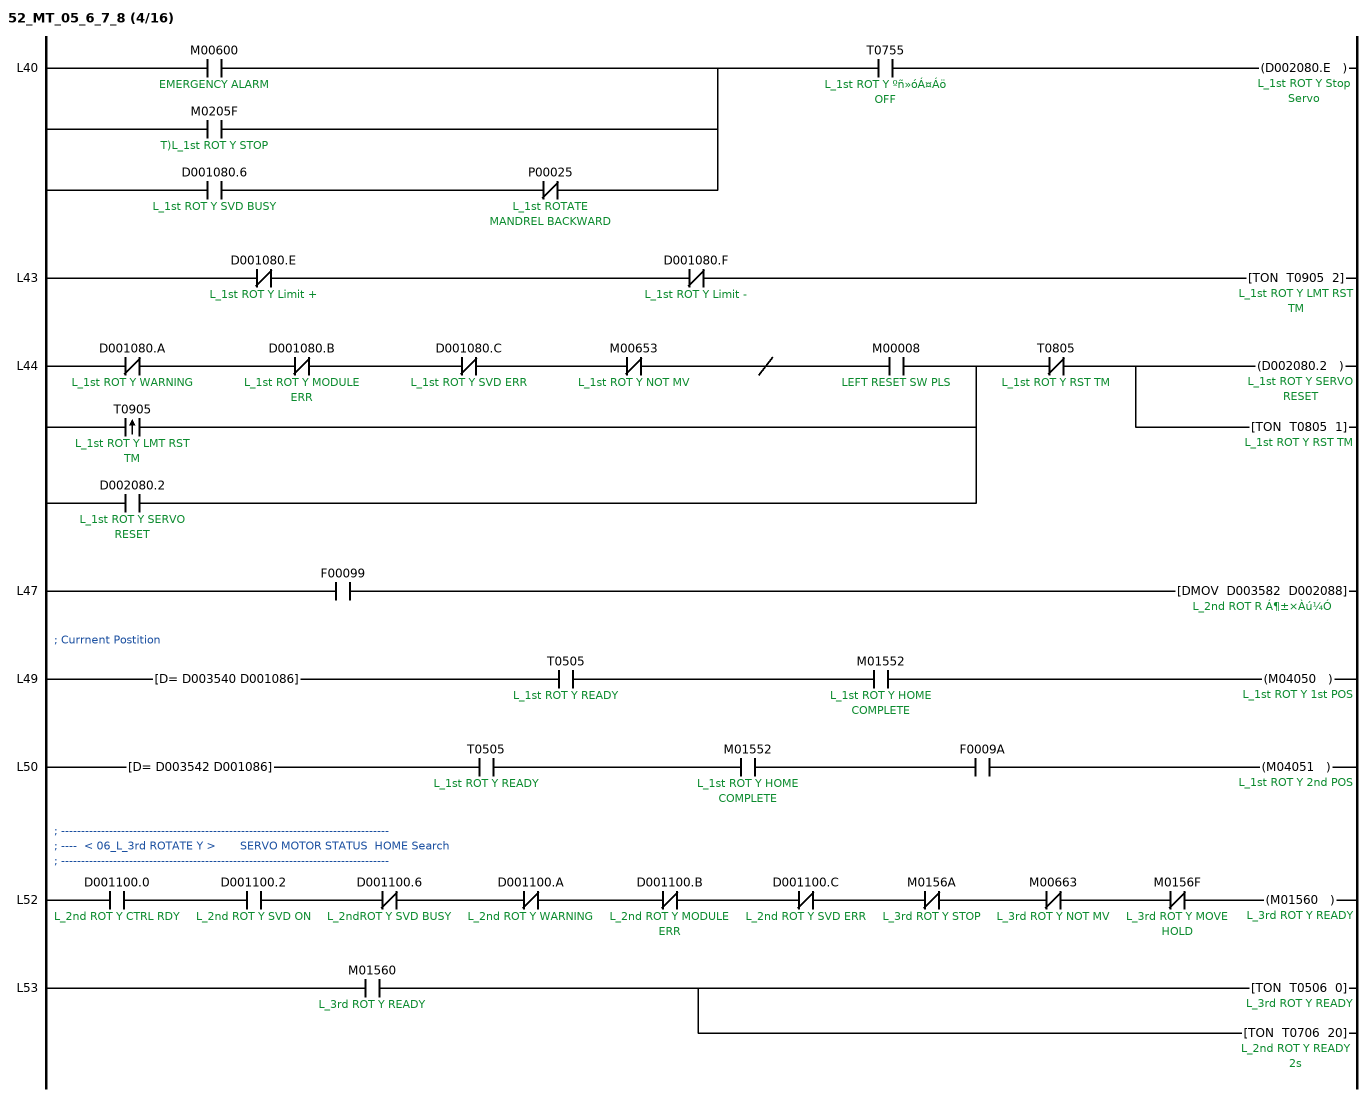
[picture p264: 52_MT_05_6_7_8 rungs L40-L53]
; L40
LOAD      M00600	// EMERGENCY ALARM
OR        M0205F	// T)L_1st ROT Y STOP
LOAD      D001080.6	// L_1st ROT Y SVD BUSY
AND NOT   P00025	// L_1st ROTATE MANDREL BACKWARD
OR LOAD
AND       T0755	// L_1st ROT Y ºñ»óÁ¤Áö OFF
OUT       D002080.E	// L_1st ROT Y Stop Servo
; L43
LOAD NOT  D001080.E	// L_1st ROT Y Limit +
AND NOT   D001080.F	// L_1st ROT Y Limit -
TON       T0905 2	// L_1st ROT Y LMT RST TM
; L44
LOAD NOT  D001080.A	// L_1st ROT Y WARNING
AND NOT   D001080.B	// L_1st ROT Y MODULE ERR
AND NOT   D001080.C	// L_1st ROT Y SVD ERR
AND NOT   M00653	// L_1st ROT Y NOT MV
NOT
AND       M00008	// LEFT RESET SW PLS
ORP       T0905	// L_1st ROT Y LMT RST TM
OR        D002080.2	// L_1st ROT Y SERVO RESET
AND NOT   T0805	// L_1st ROT Y RST TM
OUT       D002080.2	// L_1st ROT Y SERVO RESET
TON       T0805 1	// L_1st ROT Y RST TM
; L47
LOAD      F00099
DMOV      D003582 D002088	// L_2nd ROT R Á¶±×Àú¼Ó
// Currnent Postition
; L49
LOADD=    D003540 D001086
AND       T0505	// L_1st ROT Y READY
AND       M01552	// L_1st ROT Y HOME COMPLETE
OUT       M04050	// L_1st ROT Y 1st POS
; L50
LOADD=    D003542 D001086
AND       T0505	// L_1st ROT Y READY
AND       M01552	// L_1st ROT Y HOME COMPLETE
AND       F0009A
OUT       M04051	// L_1st ROT Y 2nd POS
// ----------------------------------------------------------------------------------
// 
// ----  < 06_L_3rd ROTATE Y >       SERVO MOTOR STATUS  HOME Search
// 
// ----------------------------------------------------------------------------------
; L52
LOAD      D001100.0	// L_2nd ROT Y CTRL RDY
AND       D001100.2	// L_2nd ROT Y SVD ON
AND NOT   D001100.6	// L_2ndROT Y SVD BUSY
AND NOT   D001100.A	// L_2nd ROT Y WARNING
AND NOT   D001100.B	// L_2nd ROT Y MODULE ERR
AND NOT   D001100.C	// L_2nd ROT Y SVD ERR
AND NOT   M0156A	// L_3rd ROT Y STOP
AND NOT   M00663	// L_3rd ROT Y NOT MV
AND NOT   M0156F	// L_3rd ROT Y MOVE HOLD
OUT       M01560	// L_3rd ROT Y READY
; L53
LOAD      M01560	// L_3rd ROT Y READY
TON       T0506 0	// L_3rd ROT Y READY
TON       T0706 20	// L_2nd ROT Y READY 2s

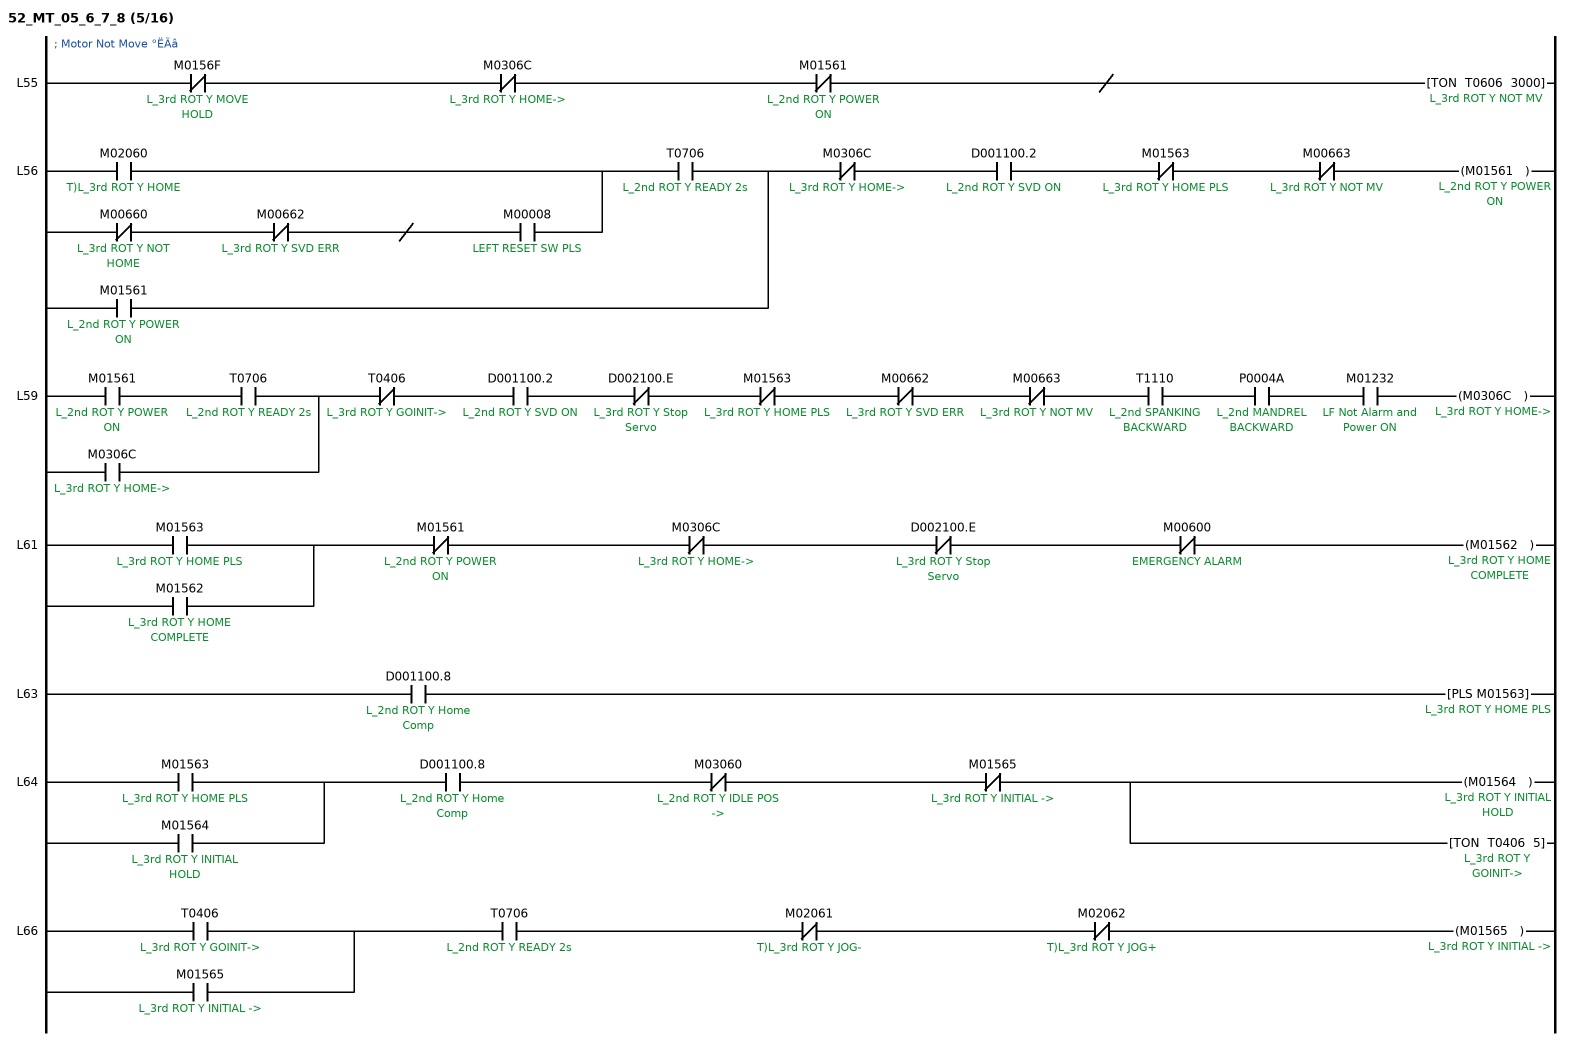
; L55
LOAD NOT  M0156F	// L_3rd ROT Y MOVE HOLD
AND NOT   M0306C	// L_3rd ROT Y HOME->
AND NOT   M01561	// L_2nd ROT Y POWER ON
NOT
TON       T0606 3000	// L_3rd ROT Y NOT MV
// output comment: Motor Not Move °ËÃâ
; L56
LOAD      M02060	// T)L_3rd ROT Y HOME
LOAD NOT  M00660	// L_3rd ROT Y NOT HOME
AND NOT   M00662	// L_3rd ROT Y SVD ERR
NOT
AND       M00008	// LEFT RESET SW PLS
OR LOAD
AND       T0706	// L_2nd ROT Y READY 2s
OR        M01561	// L_2nd ROT Y POWER ON
AND NOT   M0306C	// L_3rd ROT Y HOME->
AND       D001100.2	// L_2nd ROT Y SVD ON
AND NOT   M01563	// L_3rd ROT Y HOME PLS
AND NOT   M00663	// L_3rd ROT Y NOT MV
OUT       M01561	// L_2nd ROT Y POWER ON
; L59
LOAD      M01561	// L_2nd ROT Y POWER ON
AND       T0706	// L_2nd ROT Y READY 2s
OR        M0306C	// L_3rd ROT Y HOME->
AND NOT   T0406	// L_3rd ROT Y GOINIT->
AND       D001100.2	// L_2nd ROT Y SVD ON
AND NOT   D002100.E	// L_3rd ROT Y Stop Servo
AND NOT   M01563	// L_3rd ROT Y HOME PLS
AND NOT   M00662	// L_3rd ROT Y SVD ERR
AND NOT   M00663	// L_3rd ROT Y NOT MV
AND       T1110	// L_2nd SPANKING BACKWARD
AND       P0004A	// L_2nd MANDREL BACKWARD
AND       M01232	// LF Not Alarm and Power ON
OUT       M0306C	// L_3rd ROT Y HOME->
; L61
LOAD      M01563	// L_3rd ROT Y HOME PLS
OR        M01562	// L_3rd ROT Y HOME COMPLETE
AND NOT   M01561	// L_2nd ROT Y POWER ON
AND NOT   M0306C	// L_3rd ROT Y HOME->
AND NOT   D002100.E	// L_3rd ROT Y Stop Servo
AND NOT   M00600	// EMERGENCY ALARM
OUT       M01562	// L_3rd ROT Y HOME COMPLETE
; L63
LOAD      D001100.8	// L_2nd ROT Y Home Comp
OUTP      M01563	// L_3rd ROT Y HOME PLS
; L64
LOAD      M01563	// L_3rd ROT Y HOME PLS
OR        M01564	// L_3rd ROT Y INITIAL HOLD
AND       D001100.8	// L_2nd ROT Y Home Comp
AND NOT   M03060	// L_2nd ROT Y IDLE POS ->
AND NOT   M01565	// L_3rd ROT Y INITIAL ->
OUT       M01564	// L_3rd ROT Y INITIAL HOLD
TON       T0406 5	// L_3rd ROT Y GOINIT->
; L66
LOAD      T0406	// L_3rd ROT Y GOINIT->
OR        M01565	// L_3rd ROT Y INITIAL ->
AND       T0706	// L_2nd ROT Y READY 2s
AND NOT   M02061	// T)L_3rd ROT Y JOG-
AND NOT   M02062	// T)L_3rd ROT Y JOG+
OUT       M01565	// L_3rd ROT Y INITIAL ->

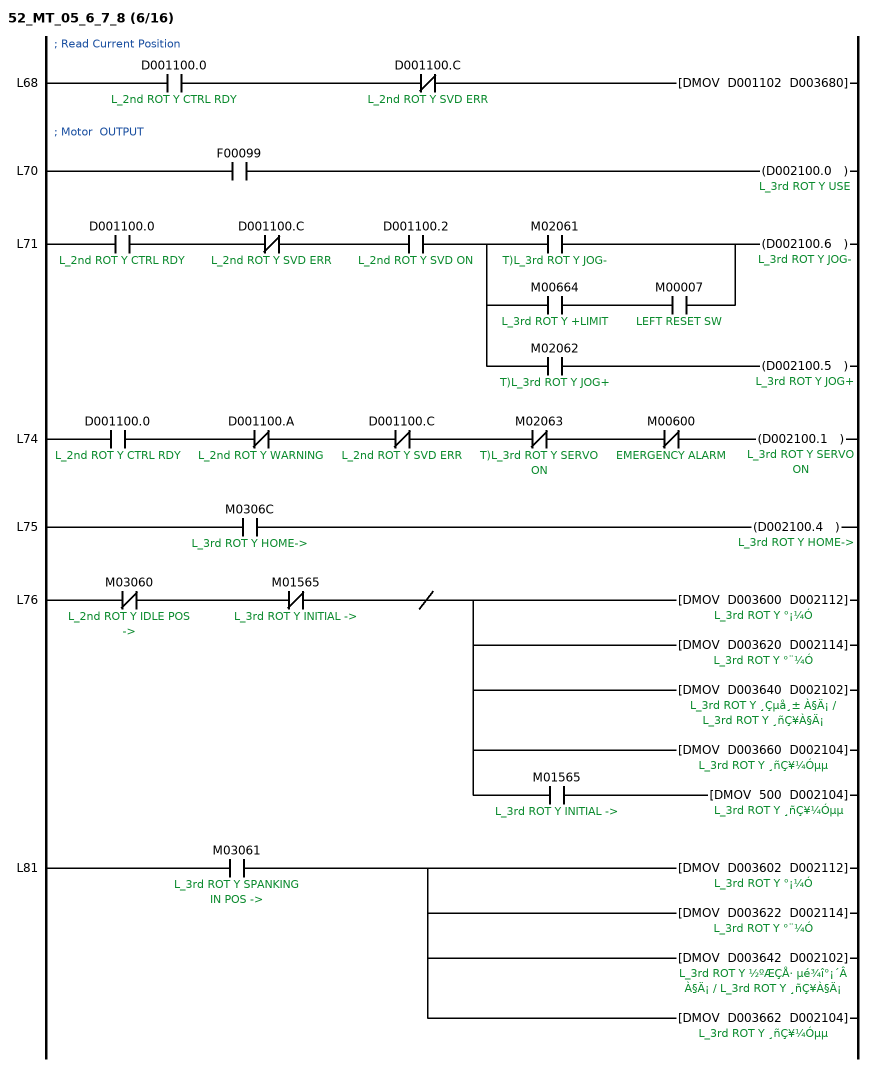
; L68
LOAD      D001100.0	// L_2nd ROT Y CTRL RDY
AND NOT   D001100.C	// L_2nd ROT Y SVD ERR
DMOV      D001102 D003680
// output comment: Read Current Position
//  Motor  OUTPUT
; L70
LOAD      F00099
OUT       D002100.0	// L_3rd ROT Y USE
; L71
LOAD      D001100.0	// L_2nd ROT Y CTRL RDY
AND NOT   D001100.C	// L_2nd ROT Y SVD ERR
AND       D001100.2	// L_2nd ROT Y SVD ON
MPUSH
LOAD      M02061	// T)L_3rd ROT Y JOG-
LOAD      M00664	// L_3rd ROT Y +LIMIT
AND       M00007	// LEFT RESET SW
OR LOAD
AND LOAD
OUT       D002100.6	// L_3rd ROT Y JOG-
MPOP
AND       M02062	// T)L_3rd ROT Y JOG+
OUT       D002100.5	// L_3rd ROT Y JOG+
; L74
LOAD      D001100.0	// L_2nd ROT Y CTRL RDY
AND NOT   D001100.A	// L_2nd ROT Y WARNING
AND NOT   D001100.C	// L_2nd ROT Y SVD ERR
AND NOT   M02063	// T)L_3rd ROT Y SERVO ON
AND NOT   M00600	// EMERGENCY ALARM
OUT       D002100.1	// L_3rd ROT Y SERVO ON
; L75
LOAD      M0306C	// L_3rd ROT Y HOME->
OUT       D002100.4	// L_3rd ROT Y HOME->
; L76
LOAD NOT  M03060	// L_2nd ROT Y IDLE POS ->
AND NOT   M01565	// L_3rd ROT Y INITIAL ->
NOT
DMOV      D003600 D002112	// L_3rd ROT Y °¡¼Ó
DMOV      D003620 D002114	// L_3rd ROT Y °¨¼Ó
DMOV      D003640 D002102	// L_3rd ROT Y ¸Çµå¸± À§Ä¡ / L_3rd ROT Y ¸ñÇ¥À§Ä¡
DMOV      D003660 D002104	// L_3rd ROT Y ¸ñÇ¥¼Óµµ
AND       M01565	// L_3rd ROT Y INITIAL ->
DMOV      500 D002104	// L_3rd ROT Y ¸ñÇ¥¼Óµµ
; L81
LOAD      M03061	// L_3rd ROT Y SPANKING IN POS ->
DMOV      D003602 D002112	// L_3rd ROT Y °¡¼Ó
DMOV      D003622 D002114	// L_3rd ROT Y °¨¼Ó
DMOV      D003642 D002102	// L_3rd ROT Y ½ºÆÇÅ· µé¾î°¡´Â À§Ä¡ / L_3rd ROT Y ¸ñÇ¥À§Ä¡
DMOV      D003662 D002104	// L_3rd ROT Y ¸ñÇ¥¼Óµµ

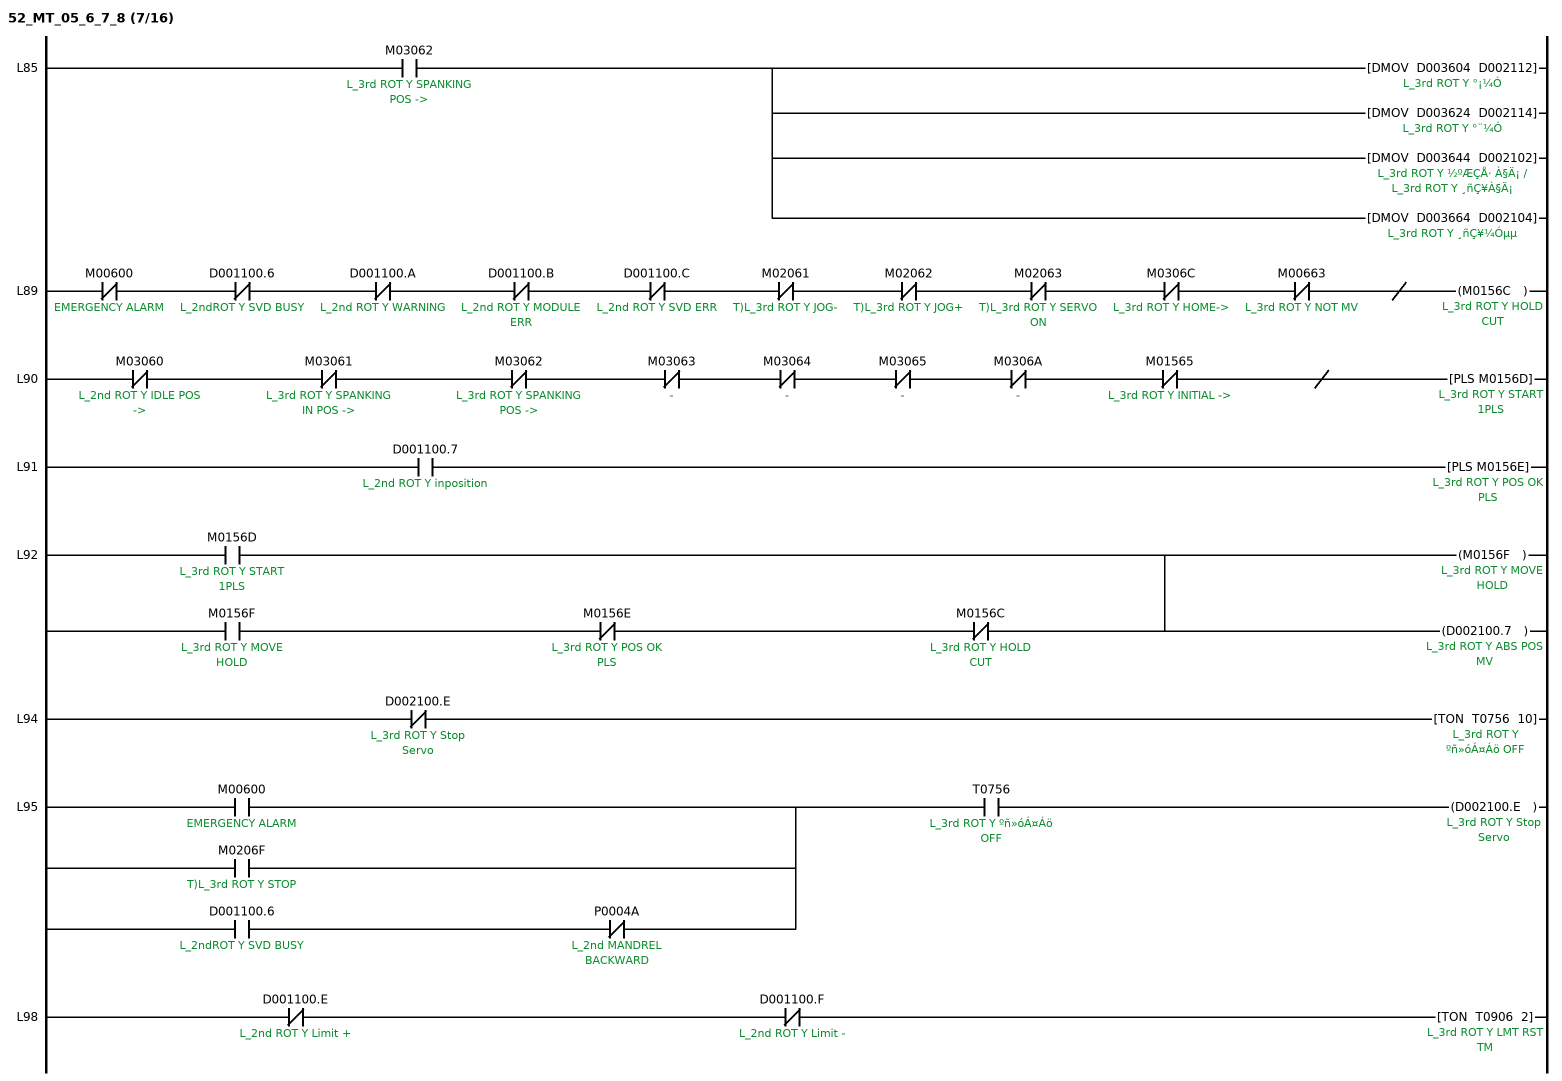
; L85
LOAD      M03062	// L_3rd ROT Y SPANKING POS ->
DMOV      D003604 D002112	// L_3rd ROT Y °¡¼Ó
DMOV      D003624 D002114	// L_3rd ROT Y °¨¼Ó
DMOV      D003644 D002102	// L_3rd ROT Y ½ºÆÇÅ· À§Ä¡ / L_3rd ROT Y ¸ñÇ¥À§Ä¡
DMOV      D003664 D002104	// L_3rd ROT Y ¸ñÇ¥¼Óµµ
; L89
LOAD NOT  M00600	// EMERGENCY ALARM
AND NOT   D001100.6	// L_2ndROT Y SVD BUSY
AND NOT   D001100.A	// L_2nd ROT Y WARNING
AND NOT   D001100.B	// L_2nd ROT Y MODULE ERR
AND NOT   D001100.C	// L_2nd ROT Y SVD ERR
AND NOT   M02061	// T)L_3rd ROT Y JOG-
AND NOT   M02062	// T)L_3rd ROT Y JOG+
AND NOT   M02063	// T)L_3rd ROT Y SERVO ON
AND NOT   M0306C	// L_3rd ROT Y HOME->
AND NOT   M00663	// L_3rd ROT Y NOT MV
NOT
OUT       M0156C	// L_3rd ROT Y HOLD CUT
; L90
LOAD NOT  M03060	// L_2nd ROT Y IDLE POS ->
AND NOT   M03061	// L_3rd ROT Y SPANKING IN POS ->
AND NOT   M03062	// L_3rd ROT Y SPANKING POS ->
AND NOT   M03063	// -
AND NOT   M03064	// -
AND NOT   M03065	// -
AND NOT   M0306A	// -
AND NOT   M01565	// L_3rd ROT Y INITIAL ->
NOT
OUTP      M0156D	// L_3rd ROT Y START 1PLS
; L91
LOAD      D001100.7	// L_2nd ROT Y inposition
OUTP      M0156E	// L_3rd ROT Y POS OK PLS
; L92
LOAD      M0156D	// L_3rd ROT Y START 1PLS
LOAD      M0156F	// L_3rd ROT Y MOVE HOLD
AND NOT   M0156E	// L_3rd ROT Y POS OK PLS
AND NOT   M0156C	// L_3rd ROT Y HOLD CUT
OR LOAD
OUT       M0156F	// L_3rd ROT Y MOVE HOLD
OUT       D002100.7	// L_3rd ROT Y ABS POS MV
; L94
LOAD NOT  D002100.E	// L_3rd ROT Y Stop Servo
TON       T0756 10	// L_3rd ROT Y ºñ»óÁ¤Áö OFF
; L95
LOAD      M00600	// EMERGENCY ALARM
OR        M0206F	// T)L_3rd ROT Y STOP
LOAD      D001100.6	// L_2ndROT Y SVD BUSY
AND NOT   P0004A	// L_2nd MANDREL BACKWARD
OR LOAD
AND       T0756	// L_3rd ROT Y ºñ»óÁ¤Áö OFF
OUT       D002100.E	// L_3rd ROT Y Stop Servo
; L98
LOAD NOT  D001100.E	// L_2nd ROT Y Limit +
AND NOT   D001100.F	// L_2nd ROT Y Limit -
TON       T0906 2	// L_3rd ROT Y LMT RST TM

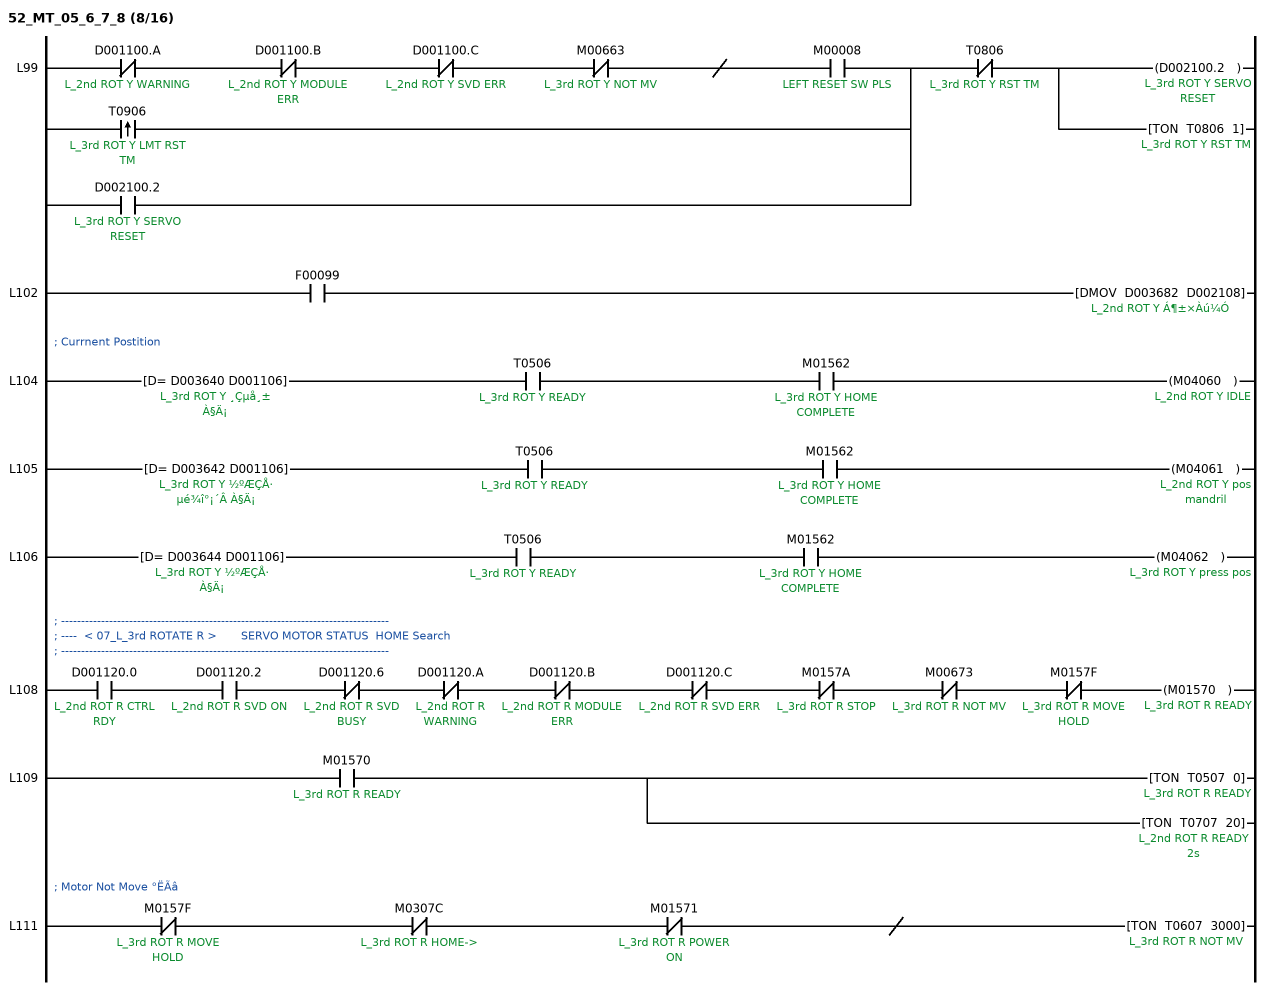
; L99
LOAD NOT  D001100.A	// L_2nd ROT Y WARNING
AND NOT   D001100.B	// L_2nd ROT Y MODULE ERR
AND NOT   D001100.C	// L_2nd ROT Y SVD ERR
AND NOT   M00663	// L_3rd ROT Y NOT MV
NOT
AND       M00008	// LEFT RESET SW PLS
ORP       T0906	// L_3rd ROT Y LMT RST TM
OR        D002100.2	// L_3rd ROT Y SERVO RESET
AND NOT   T0806	// L_3rd ROT Y RST TM
OUT       D002100.2	// L_3rd ROT Y SERVO RESET
TON       T0806 1	// L_3rd ROT Y RST TM
; L102
LOAD      F00099
DMOV      D003682 D002108	// L_2nd ROT Y Á¶±×Àú¼Ó
// Currnent Postition
; L104
LOADD=    D003640 D001106	// L_3rd ROT Y ¸Çµå¸± À§Ä¡
AND       T0506	// L_3rd ROT Y READY
AND       M01562	// L_3rd ROT Y HOME COMPLETE
OUT       M04060	// L_2nd ROT Y IDLE
; L105
LOADD=    D003642 D001106	// L_3rd ROT Y ½ºÆÇÅ· µé¾î°¡´Â À§Ä¡
AND       T0506	// L_3rd ROT Y READY
AND       M01562	// L_3rd ROT Y HOME COMPLETE
OUT       M04061	// L_2nd ROT Y pos mandril
; L106
LOADD=    D003644 D001106	// L_3rd ROT Y ½ºÆÇÅ· À§Ä¡
AND       T0506	// L_3rd ROT Y READY
AND       M01562	// L_3rd ROT Y HOME COMPLETE
OUT       M04062	// L_3rd ROT Y press pos
// ----------------------------------------------------------------------------------
// 
// ----  < 07_L_3rd ROTATE R >       SERVO MOTOR STATUS  HOME Search
// 
// ----------------------------------------------------------------------------------
; L108
LOAD      D001120.0	// L_2nd ROT R CTRL RDY
AND       D001120.2	// L_2nd ROT R SVD ON
AND NOT   D001120.6	// L_2nd ROT R SVD BUSY
AND NOT   D001120.A	// L_2nd ROT R WARNING
AND NOT   D001120.B	// L_2nd ROT R MODULE ERR
AND NOT   D001120.C	// L_2nd ROT R SVD ERR
AND NOT   M0157A	// L_3rd ROT R STOP
AND NOT   M00673	// L_3rd ROT R NOT MV
AND NOT   M0157F	// L_3rd ROT R MOVE HOLD
OUT       M01570	// L_3rd ROT R READY
; L109
LOAD      M01570	// L_3rd ROT R READY
TON       T0507 0	// L_3rd ROT R READY
TON       T0707 20	// L_2nd ROT R READY 2s
; L111
LOAD NOT  M0157F	// L_3rd ROT R MOVE HOLD
AND NOT   M0307C	// L_3rd ROT R HOME->
AND NOT   M01571	// L_3rd ROT R POWER ON
NOT
TON       T0607 3000	// L_3rd ROT R NOT MV
// output comment: Motor Not Move °ËÃâ

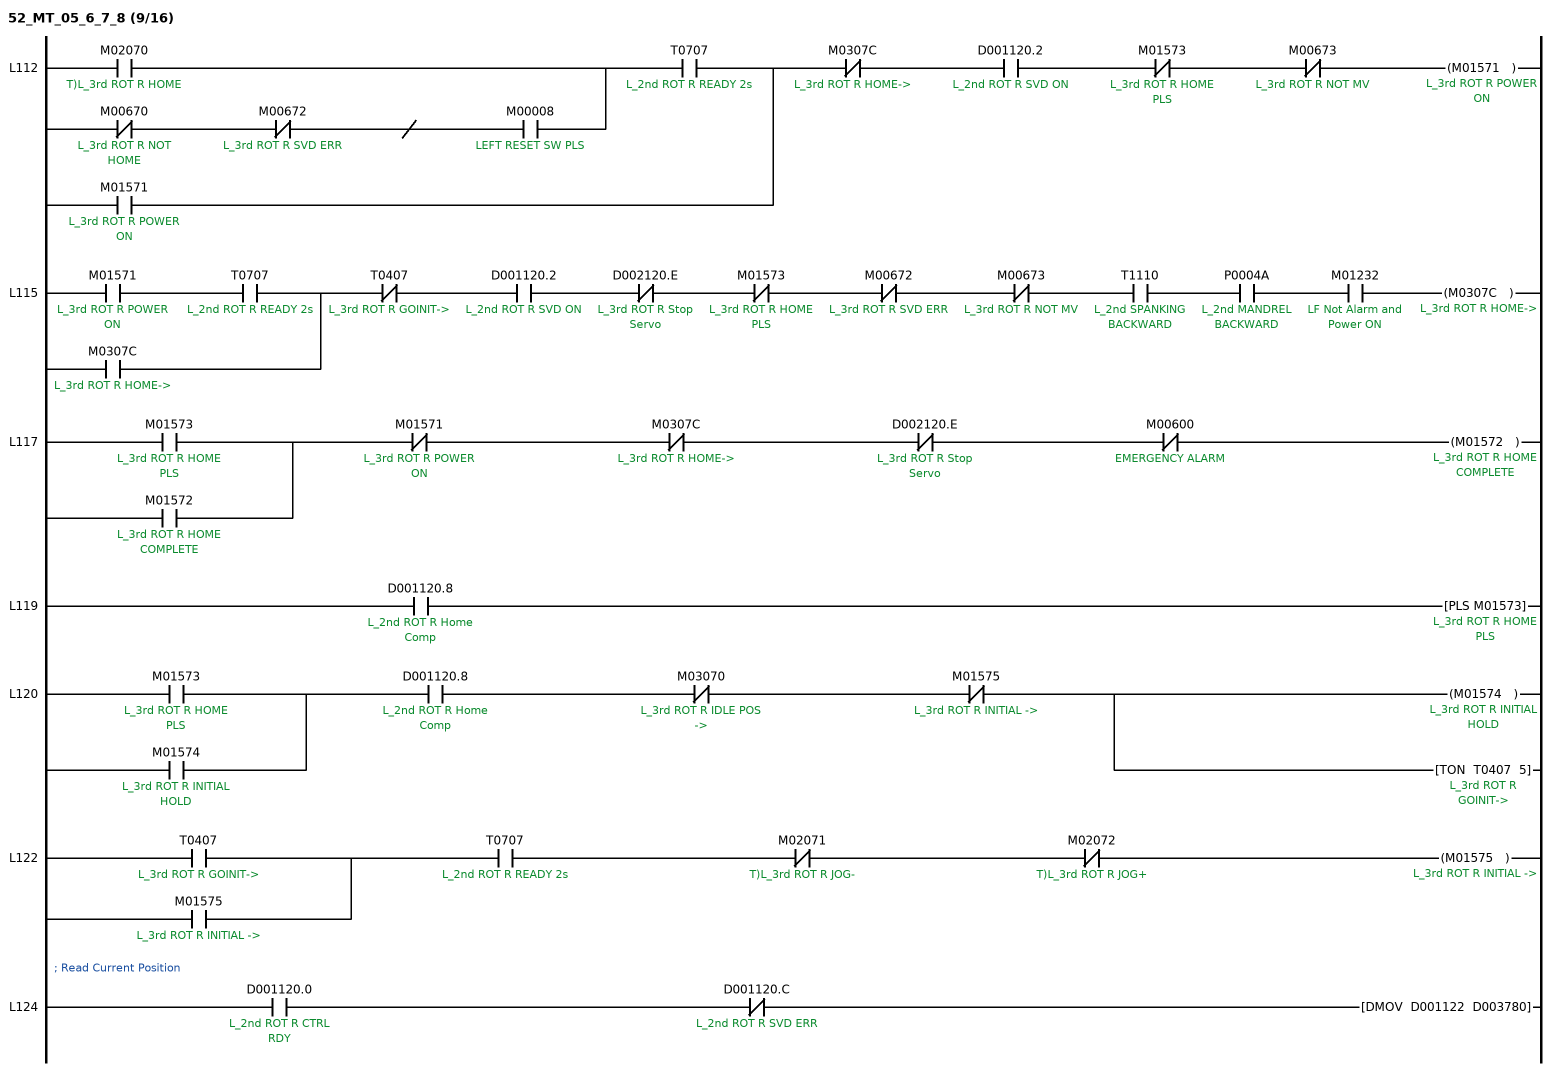
; L112
LOAD      M02070	// T)L_3rd ROT R HOME
LOAD NOT  M00670	// L_3rd ROT R NOT HOME
AND NOT   M00672	// L_3rd ROT R SVD ERR
NOT
AND       M00008	// LEFT RESET SW PLS
OR LOAD
AND       T0707	// L_2nd ROT R READY 2s
OR        M01571	// L_3rd ROT R POWER ON
AND NOT   M0307C	// L_3rd ROT R HOME->
AND       D001120.2	// L_2nd ROT R SVD ON
AND NOT   M01573	// L_3rd ROT R HOME PLS
AND NOT   M00673	// L_3rd ROT R NOT MV
OUT       M01571	// L_3rd ROT R POWER ON
; L115
LOAD      M01571	// L_3rd ROT R POWER ON
AND       T0707	// L_2nd ROT R READY 2s
OR        M0307C	// L_3rd ROT R HOME->
AND NOT   T0407	// L_3rd ROT R GOINIT->
AND       D001120.2	// L_2nd ROT R SVD ON
AND NOT   D002120.E	// L_3rd ROT R Stop Servo
AND NOT   M01573	// L_3rd ROT R HOME PLS
AND NOT   M00672	// L_3rd ROT R SVD ERR
AND NOT   M00673	// L_3rd ROT R NOT MV
AND       T1110	// L_2nd SPANKING BACKWARD
AND       P0004A	// L_2nd MANDREL BACKWARD
AND       M01232	// LF Not Alarm and Power ON
OUT       M0307C	// L_3rd ROT R HOME->
; L117
LOAD      M01573	// L_3rd ROT R HOME PLS
OR        M01572	// L_3rd ROT R HOME COMPLETE
AND NOT   M01571	// L_3rd ROT R POWER ON
AND NOT   M0307C	// L_3rd ROT R HOME->
AND NOT   D002120.E	// L_3rd ROT R Stop Servo
AND NOT   M00600	// EMERGENCY ALARM
OUT       M01572	// L_3rd ROT R HOME COMPLETE
; L119
LOAD      D001120.8	// L_2nd ROT R Home Comp
OUTP      M01573	// L_3rd ROT R HOME PLS
; L120
LOAD      M01573	// L_3rd ROT R HOME PLS
OR        M01574	// L_3rd ROT R INITIAL HOLD
AND       D001120.8	// L_2nd ROT R Home Comp
AND NOT   M03070	// L_3rd ROT R IDLE POS ->
AND NOT   M01575	// L_3rd ROT R INITIAL ->
OUT       M01574	// L_3rd ROT R INITIAL HOLD
TON       T0407 5	// L_3rd ROT R GOINIT->
; L122
LOAD      T0407	// L_3rd ROT R GOINIT->
OR        M01575	// L_3rd ROT R INITIAL ->
AND       T0707	// L_2nd ROT R READY 2s
AND NOT   M02071	// T)L_3rd ROT R JOG-
AND NOT   M02072	// T)L_3rd ROT R JOG+
OUT       M01575	// L_3rd ROT R INITIAL ->
; L124
LOAD      D001120.0	// L_2nd ROT R CTRL RDY
AND NOT   D001120.C	// L_2nd ROT R SVD ERR
DMOV      D001122 D003780
// output comment: Read Current Position

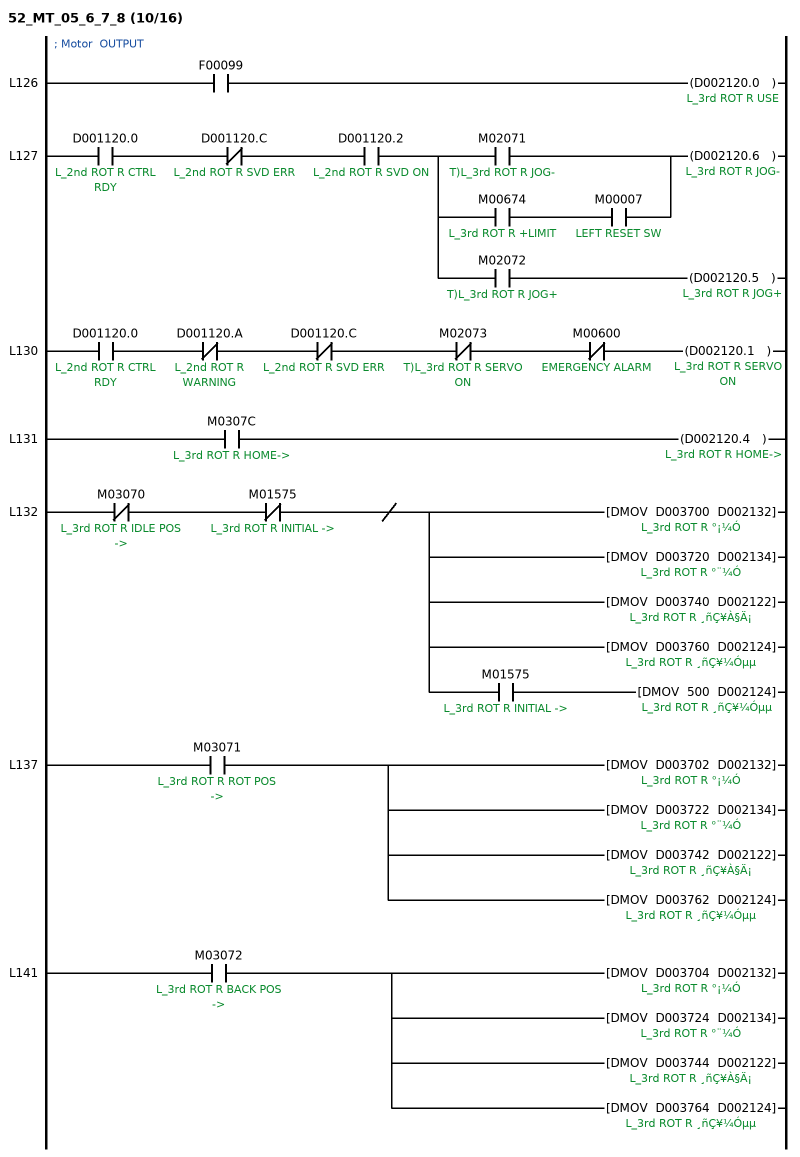
//  Motor  OUTPUT
; L126
LOAD      F00099
OUT       D002120.0	// L_3rd ROT R USE
; L127
LOAD      D001120.0	// L_2nd ROT R CTRL RDY
AND NOT   D001120.C	// L_2nd ROT R SVD ERR
AND       D001120.2	// L_2nd ROT R SVD ON
MPUSH
LOAD      M02071	// T)L_3rd ROT R JOG-
LOAD      M00674	// L_3rd ROT R +LIMIT
AND       M00007	// LEFT RESET SW
OR LOAD
AND LOAD
OUT       D002120.6	// L_3rd ROT R JOG-
MPOP
AND       M02072	// T)L_3rd ROT R JOG+
OUT       D002120.5	// L_3rd ROT R JOG+
; L130
LOAD      D001120.0	// L_2nd ROT R CTRL RDY
AND NOT   D001120.A	// L_2nd ROT R WARNING
AND NOT   D001120.C	// L_2nd ROT R SVD ERR
AND NOT   M02073	// T)L_3rd ROT R SERVO ON
AND NOT   M00600	// EMERGENCY ALARM
OUT       D002120.1	// L_3rd ROT R SERVO ON
; L131
LOAD      M0307C	// L_3rd ROT R HOME->
OUT       D002120.4	// L_3rd ROT R HOME->
; L132
LOAD NOT  M03070	// L_3rd ROT R IDLE POS ->
AND NOT   M01575	// L_3rd ROT R INITIAL ->
NOT
DMOV      D003700 D002132	// L_3rd ROT R °¡¼Ó
DMOV      D003720 D002134	// L_3rd ROT R °¨¼Ó
DMOV      D003740 D002122	// L_3rd ROT R ¸ñÇ¥À§Ä¡
DMOV      D003760 D002124	// L_3rd ROT R ¸ñÇ¥¼Óµµ
AND       M01575	// L_3rd ROT R INITIAL ->
DMOV      500 D002124	// L_3rd ROT R ¸ñÇ¥¼Óµµ
; L137
LOAD      M03071	// L_3rd ROT R ROT POS ->
DMOV      D003702 D002132	// L_3rd ROT R °¡¼Ó
DMOV      D003722 D002134	// L_3rd ROT R °¨¼Ó
DMOV      D003742 D002122	// L_3rd ROT R ¸ñÇ¥À§Ä¡
DMOV      D003762 D002124	// L_3rd ROT R ¸ñÇ¥¼Óµµ
; L141
LOAD      M03072	// L_3rd ROT R BACK POS ->
DMOV      D003704 D002132	// L_3rd ROT R °¡¼Ó
DMOV      D003724 D002134	// L_3rd ROT R °¨¼Ó
DMOV      D003744 D002122	// L_3rd ROT R ¸ñÇ¥À§Ä¡
DMOV      D003764 D002124	// L_3rd ROT R ¸ñÇ¥¼Óµµ

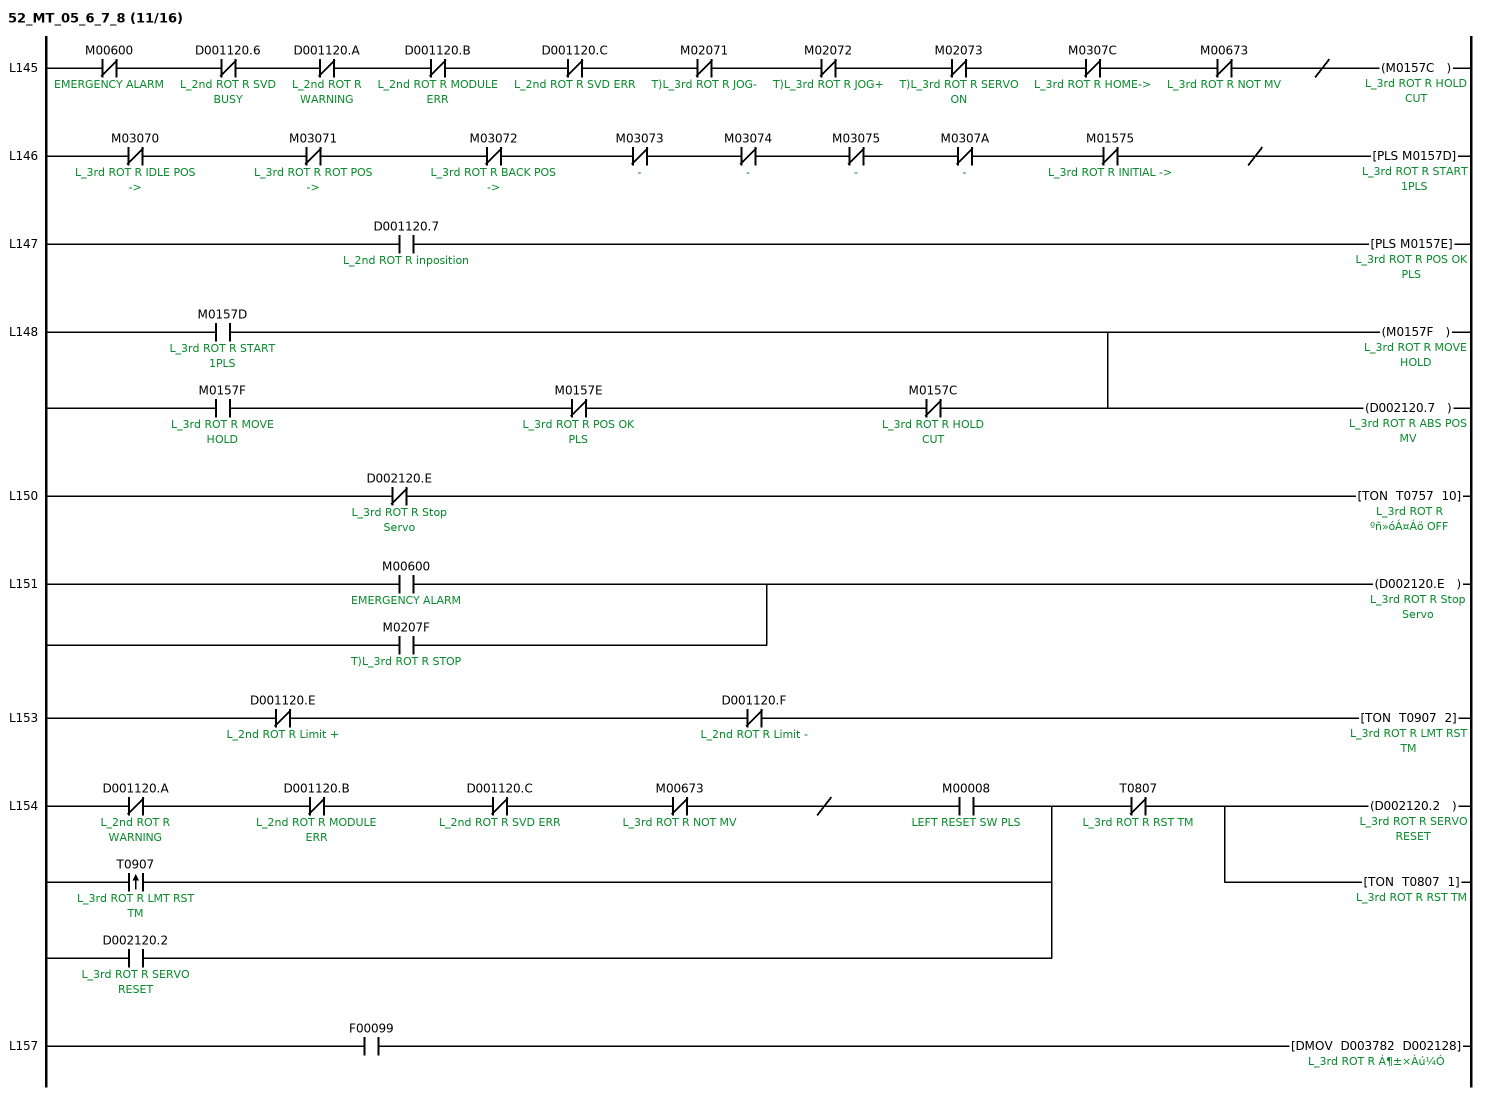
; L145
LOAD NOT  M00600	// EMERGENCY ALARM
AND NOT   D001120.6	// L_2nd ROT R SVD BUSY
AND NOT   D001120.A	// L_2nd ROT R WARNING
AND NOT   D001120.B	// L_2nd ROT R MODULE ERR
AND NOT   D001120.C	// L_2nd ROT R SVD ERR
AND NOT   M02071	// T)L_3rd ROT R JOG-
AND NOT   M02072	// T)L_3rd ROT R JOG+
AND NOT   M02073	// T)L_3rd ROT R SERVO ON
AND NOT   M0307C	// L_3rd ROT R HOME->
AND NOT   M00673	// L_3rd ROT R NOT MV
NOT
OUT       M0157C	// L_3rd ROT R HOLD CUT
; L146
LOAD NOT  M03070	// L_3rd ROT R IDLE POS ->
AND NOT   M03071	// L_3rd ROT R ROT POS ->
AND NOT   M03072	// L_3rd ROT R BACK POS ->
AND NOT   M03073	// -
AND NOT   M03074	// -
AND NOT   M03075	// -
AND NOT   M0307A	// -
AND NOT   M01575	// L_3rd ROT R INITIAL ->
NOT
OUTP      M0157D	// L_3rd ROT R START 1PLS
; L147
LOAD      D001120.7	// L_2nd ROT R inposition
OUTP      M0157E	// L_3rd ROT R POS OK PLS
; L148
LOAD      M0157D	// L_3rd ROT R START 1PLS
LOAD      M0157F	// L_3rd ROT R MOVE HOLD
AND NOT   M0157E	// L_3rd ROT R POS OK PLS
AND NOT   M0157C	// L_3rd ROT R HOLD CUT
OR LOAD
OUT       M0157F	// L_3rd ROT R MOVE HOLD
OUT       D002120.7	// L_3rd ROT R ABS POS MV
; L150
LOAD NOT  D002120.E	// L_3rd ROT R Stop Servo
TON       T0757 10	// L_3rd ROT R ºñ»óÁ¤Áö OFF
; L151
LOAD      M00600	// EMERGENCY ALARM
OR        M0207F	// T)L_3rd ROT R STOP
OUT       D002120.E	// L_3rd ROT R Stop Servo
; L153
LOAD NOT  D001120.E	// L_2nd ROT R Limit +
AND NOT   D001120.F	// L_2nd ROT R Limit -
TON       T0907 2	// L_3rd ROT R LMT RST TM
; L154
LOAD NOT  D001120.A	// L_2nd ROT R WARNING
AND NOT   D001120.B	// L_2nd ROT R MODULE ERR
AND NOT   D001120.C	// L_2nd ROT R SVD ERR
AND NOT   M00673	// L_3rd ROT R NOT MV
NOT
AND       M00008	// LEFT RESET SW PLS
ORP       T0907	// L_3rd ROT R LMT RST TM
OR        D002120.2	// L_3rd ROT R SERVO RESET
AND NOT   T0807	// L_3rd ROT R RST TM
OUT       D002120.2	// L_3rd ROT R SERVO RESET
TON       T0807 1	// L_3rd ROT R RST TM
; L157
LOAD      F00099
DMOV      D003782 D002128	// L_3rd ROT R Á¶±×Àú¼Ó

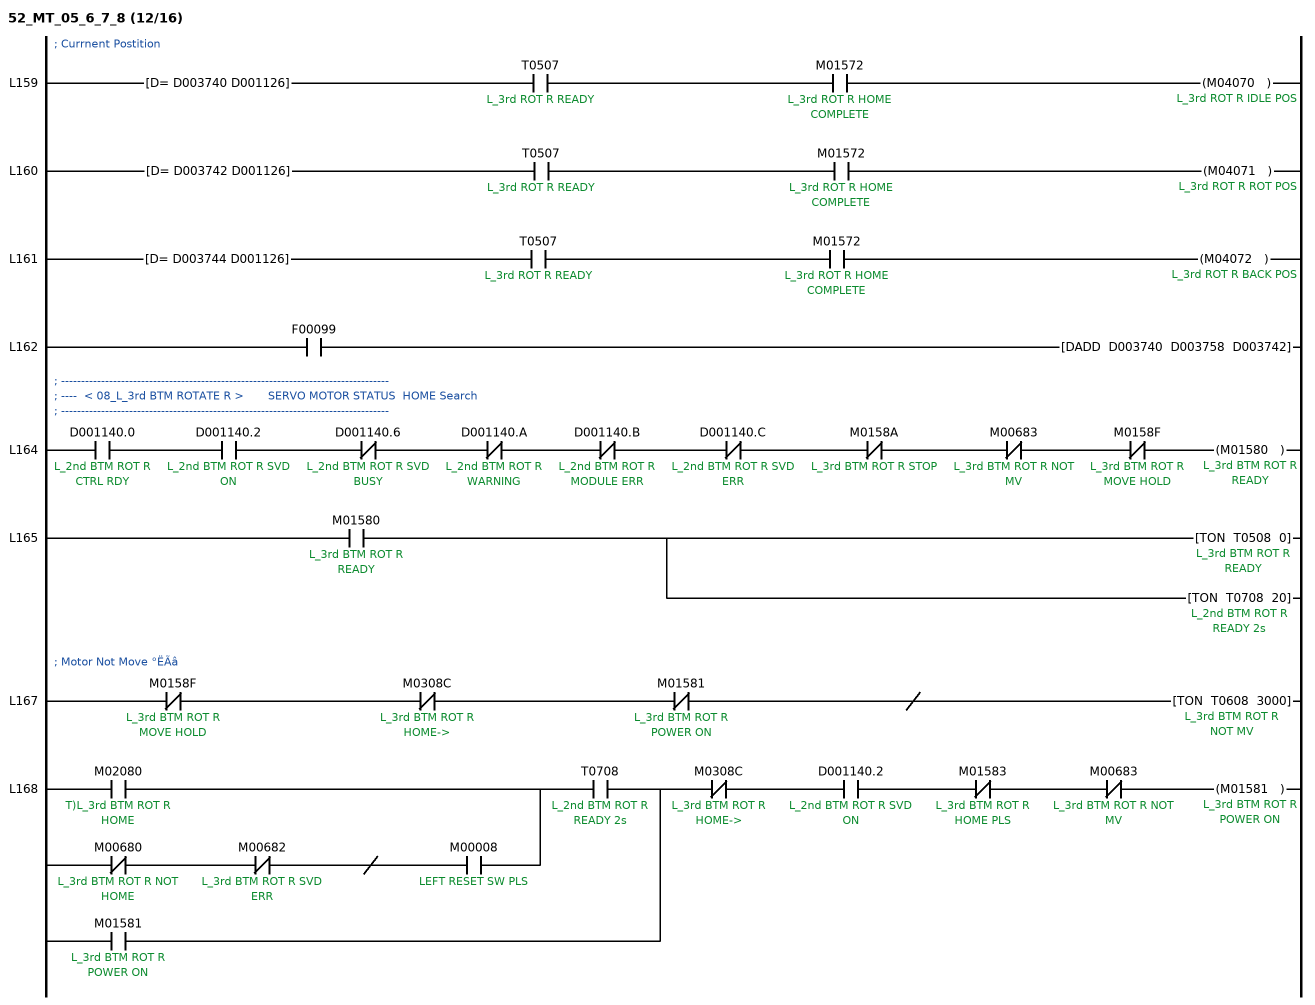
// Currnent Postition
; L159
LOADD=    D003740 D001126
AND       T0507	// L_3rd ROT R READY
AND       M01572	// L_3rd ROT R HOME COMPLETE
OUT       M04070	// L_3rd ROT R IDLE POS
; L160
LOADD=    D003742 D001126
AND       T0507	// L_3rd ROT R READY
AND       M01572	// L_3rd ROT R HOME COMPLETE
OUT       M04071	// L_3rd ROT R ROT POS
; L161
LOADD=    D003744 D001126
AND       T0507	// L_3rd ROT R READY
AND       M01572	// L_3rd ROT R HOME COMPLETE
OUT       M04072	// L_3rd ROT R BACK POS
; L162
LOAD      F00099
DADD      D003740 D003758 D003742
// ----------------------------------------------------------------------------------
// 
// ----  < 08_L_3rd BTM ROTATE R >       SERVO MOTOR STATUS  HOME Search
// 
// ----------------------------------------------------------------------------------
; L164
LOAD      D001140.0	// L_2nd BTM ROT R CTRL RDY
AND       D001140.2	// L_2nd BTM ROT R SVD ON
AND NOT   D001140.6	// L_2nd BTM ROT R SVD BUSY
AND NOT   D001140.A	// L_2nd BTM ROT R WARNING
AND NOT   D001140.B	// L_2nd BTM ROT R MODULE ERR
AND NOT   D001140.C	// L_2nd BTM ROT R SVD ERR
AND NOT   M0158A	// L_3rd BTM ROT R STOP
AND NOT   M00683	// L_3rd BTM ROT R NOT MV
AND NOT   M0158F	// L_3rd BTM ROT R MOVE HOLD
OUT       M01580	// L_3rd BTM ROT R READY
; L165
LOAD      M01580	// L_3rd BTM ROT R READY
TON       T0508 0	// L_3rd BTM ROT R READY
TON       T0708 20	// L_2nd BTM ROT R READY 2s
; L167
LOAD NOT  M0158F	// L_3rd BTM ROT R MOVE HOLD
AND NOT   M0308C	// L_3rd BTM ROT R HOME->
AND NOT   M01581	// L_3rd BTM ROT R POWER ON
NOT
TON       T0608 3000	// L_3rd BTM ROT R NOT MV
// output comment: Motor Not Move °ËÃâ
; L168
LOAD      M02080	// T)L_3rd BTM ROT R HOME
LOAD NOT  M00680	// L_3rd BTM ROT R NOT HOME
AND NOT   M00682	// L_3rd BTM ROT R SVD ERR
NOT
AND       M00008	// LEFT RESET SW PLS
OR LOAD
AND       T0708	// L_2nd BTM ROT R READY 2s
OR        M01581	// L_3rd BTM ROT R POWER ON
AND NOT   M0308C	// L_3rd BTM ROT R HOME->
AND       D001140.2	// L_2nd BTM ROT R SVD ON
AND NOT   M01583	// L_3rd BTM ROT R HOME PLS
AND NOT   M00683	// L_3rd BTM ROT R NOT MV
OUT       M01581	// L_3rd BTM ROT R POWER ON

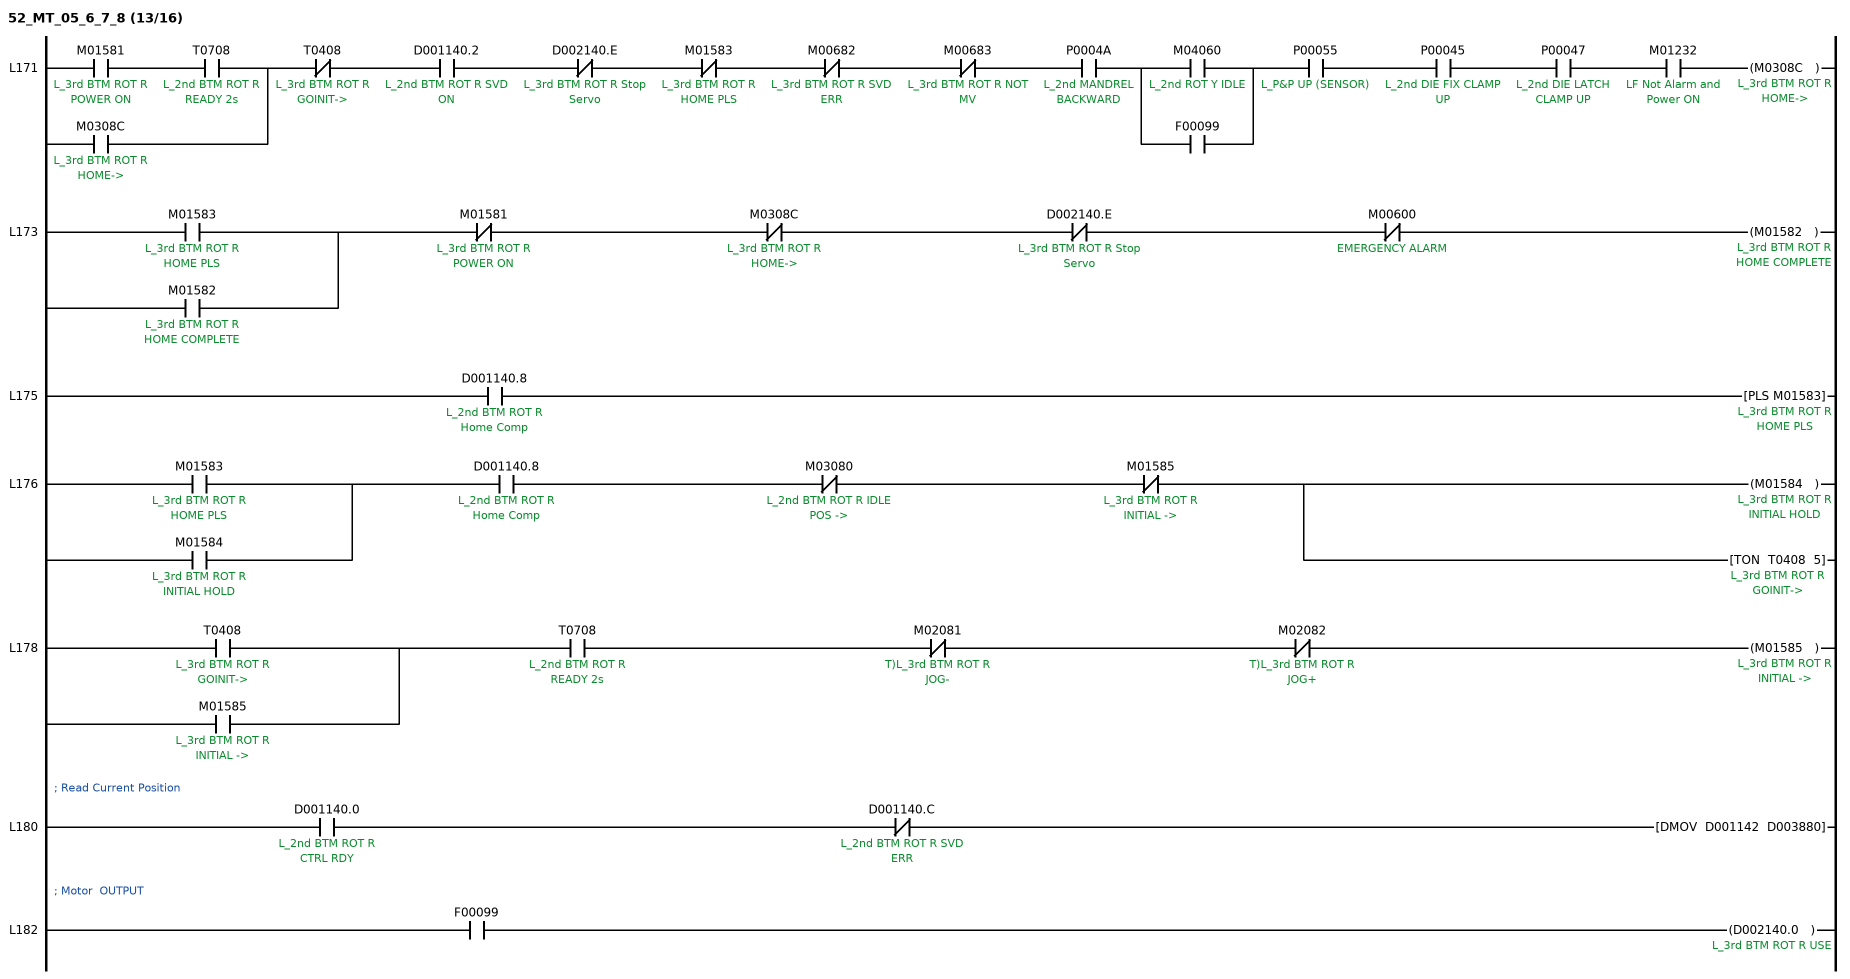
; L171
LOAD      M01581	// L_3rd BTM ROT R POWER ON
AND       T0708	// L_2nd BTM ROT R READY 2s
OR        M0308C	// L_3rd BTM ROT R HOME->
AND NOT   T0408	// L_3rd BTM ROT R GOINIT->
AND       D001140.2	// L_2nd BTM ROT R SVD ON
AND NOT   D002140.E	// L_3rd BTM ROT R Stop Servo
AND NOT   M01583	// L_3rd BTM ROT R HOME PLS
AND NOT   M00682	// L_3rd BTM ROT R SVD ERR
AND NOT   M00683	// L_3rd BTM ROT R NOT MV
AND       P0004A	// L_2nd MANDREL BACKWARD
LOAD      M04060	// L_2nd ROT Y IDLE
OR        F00099
AND LOAD
AND       P00055	// L_P&P UP (SENSOR)
AND       P00045	// L_2nd DIE FIX CLAMP UP
AND       P00047	// L_2nd DIE LATCH CLAMP UP
AND       M01232	// LF Not Alarm and Power ON
OUT       M0308C	// L_3rd BTM ROT R HOME->
; L173
LOAD      M01583	// L_3rd BTM ROT R HOME PLS
OR        M01582	// L_3rd BTM ROT R HOME COMPLETE
AND NOT   M01581	// L_3rd BTM ROT R POWER ON
AND NOT   M0308C	// L_3rd BTM ROT R HOME->
AND NOT   D002140.E	// L_3rd BTM ROT R Stop Servo
AND NOT   M00600	// EMERGENCY ALARM
OUT       M01582	// L_3rd BTM ROT R HOME COMPLETE
; L175
LOAD      D001140.8	// L_2nd BTM ROT R Home Comp
OUTP      M01583	// L_3rd BTM ROT R HOME PLS
; L176
LOAD      M01583	// L_3rd BTM ROT R HOME PLS
OR        M01584	// L_3rd BTM ROT R INITIAL HOLD
AND       D001140.8	// L_2nd BTM ROT R Home Comp
AND NOT   M03080	// L_2nd BTM ROT R IDLE POS ->
AND NOT   M01585	// L_3rd BTM ROT R INITIAL ->
OUT       M01584	// L_3rd BTM ROT R INITIAL HOLD
TON       T0408 5	// L_3rd BTM ROT R GOINIT->
; L178
LOAD      T0408	// L_3rd BTM ROT R GOINIT->
OR        M01585	// L_3rd BTM ROT R INITIAL ->
AND       T0708	// L_2nd BTM ROT R READY 2s
AND NOT   M02081	// T)L_3rd BTM ROT R JOG-
AND NOT   M02082	// T)L_3rd BTM ROT R JOG+
OUT       M01585	// L_3rd BTM ROT R INITIAL ->
; L180
LOAD      D001140.0	// L_2nd BTM ROT R CTRL RDY
AND NOT   D001140.C	// L_2nd BTM ROT R SVD ERR
DMOV      D001142 D003880
// output comment: Read Current Position
//  Motor  OUTPUT
; L182
LOAD      F00099
OUT       D002140.0	// L_3rd BTM ROT R USE

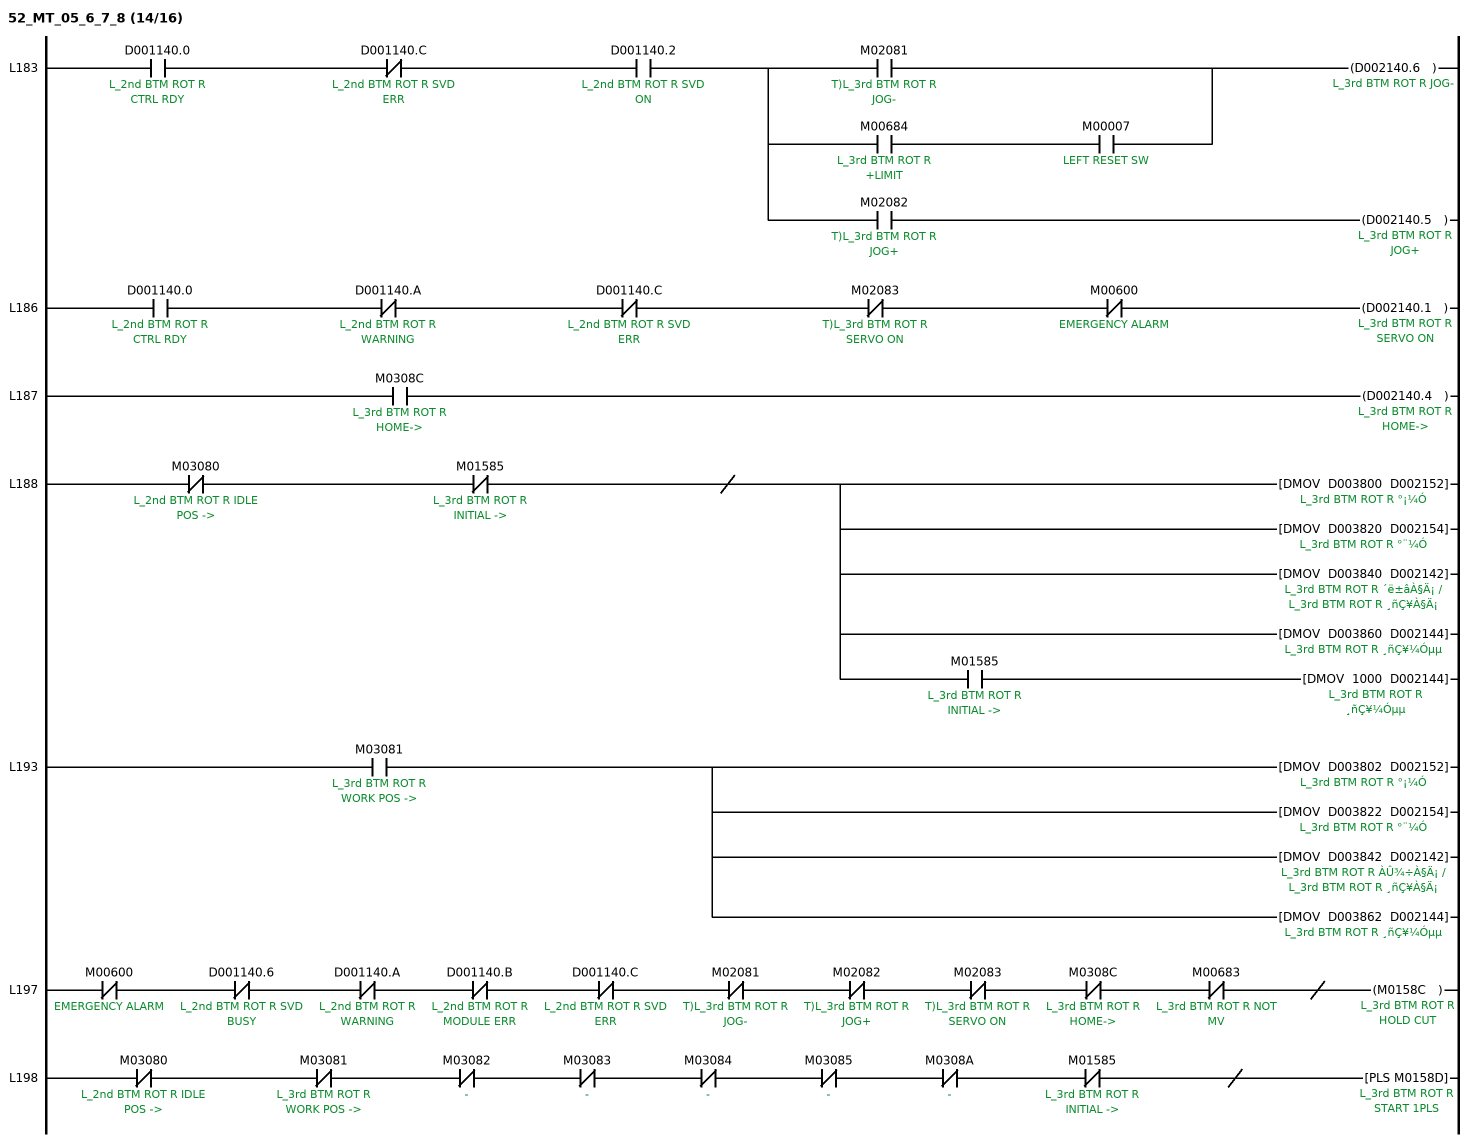
; L183
LOAD      D001140.0	// L_2nd BTM ROT R CTRL RDY
AND NOT   D001140.C	// L_2nd BTM ROT R SVD ERR
AND       D001140.2	// L_2nd BTM ROT R SVD ON
MPUSH
LOAD      M02081	// T)L_3rd BTM ROT R JOG-
LOAD      M00684	// L_3rd BTM ROT R +LIMIT
AND       M00007	// LEFT RESET SW
OR LOAD
AND LOAD
OUT       D002140.6	// L_3rd BTM ROT R JOG-
MPOP
AND       M02082	// T)L_3rd BTM ROT R JOG+
OUT       D002140.5	// L_3rd BTM ROT R JOG+
; L186
LOAD      D001140.0	// L_2nd BTM ROT R CTRL RDY
AND NOT   D001140.A	// L_2nd BTM ROT R WARNING
AND NOT   D001140.C	// L_2nd BTM ROT R SVD ERR
AND NOT   M02083	// T)L_3rd BTM ROT R SERVO ON
AND NOT   M00600	// EMERGENCY ALARM
OUT       D002140.1	// L_3rd BTM ROT R SERVO ON
; L187
LOAD      M0308C	// L_3rd BTM ROT R HOME->
OUT       D002140.4	// L_3rd BTM ROT R HOME->
; L188
LOAD NOT  M03080	// L_2nd BTM ROT R IDLE POS ->
AND NOT   M01585	// L_3rd BTM ROT R INITIAL ->
NOT
DMOV      D003800 D002152	// L_3rd BTM ROT R °¡¼Ó
DMOV      D003820 D002154	// L_3rd BTM ROT R °¨¼Ó
DMOV      D003840 D002142	// L_3rd BTM ROT R ´ë±âÀ§Ä¡ / L_3rd BTM ROT R ¸ñÇ¥À§Ä¡
DMOV      D003860 D002144	// L_3rd BTM ROT R ¸ñÇ¥¼Óµµ
AND       M01585	// L_3rd BTM ROT R INITIAL ->
DMOV      1000 D002144	// L_3rd BTM ROT R ¸ñÇ¥¼Óµµ
; L193
LOAD      M03081	// L_3rd BTM ROT R WORK POS ->
DMOV      D003802 D002152	// L_3rd BTM ROT R °¡¼Ó
DMOV      D003822 D002154	// L_3rd BTM ROT R °¨¼Ó
DMOV      D003842 D002142	// L_3rd BTM ROT R ÀÛ¾÷À§Ä¡ / L_3rd BTM ROT R ¸ñÇ¥À§Ä¡
DMOV      D003862 D002144	// L_3rd BTM ROT R ¸ñÇ¥¼Óµµ
; L197
LOAD NOT  M00600	// EMERGENCY ALARM
AND NOT   D001140.6	// L_2nd BTM ROT R SVD BUSY
AND NOT   D001140.A	// L_2nd BTM ROT R WARNING
AND NOT   D001140.B	// L_2nd BTM ROT R MODULE ERR
AND NOT   D001140.C	// L_2nd BTM ROT R SVD ERR
AND NOT   M02081	// T)L_3rd BTM ROT R JOG-
AND NOT   M02082	// T)L_3rd BTM ROT R JOG+
AND NOT   M02083	// T)L_3rd BTM ROT R SERVO ON
AND NOT   M0308C	// L_3rd BTM ROT R HOME->
AND NOT   M00683	// L_3rd BTM ROT R NOT MV
NOT
OUT       M0158C	// L_3rd BTM ROT R HOLD CUT
; L198
LOAD NOT  M03080	// L_2nd BTM ROT R IDLE POS ->
AND NOT   M03081	// L_3rd BTM ROT R WORK POS ->
AND NOT   M03082	// -
AND NOT   M03083	// -
AND NOT   M03084	// -
AND NOT   M03085	// -
AND NOT   M0308A	// -
AND NOT   M01585	// L_3rd BTM ROT R INITIAL ->
NOT
OUTP      M0158D	// L_3rd BTM ROT R START 1PLS

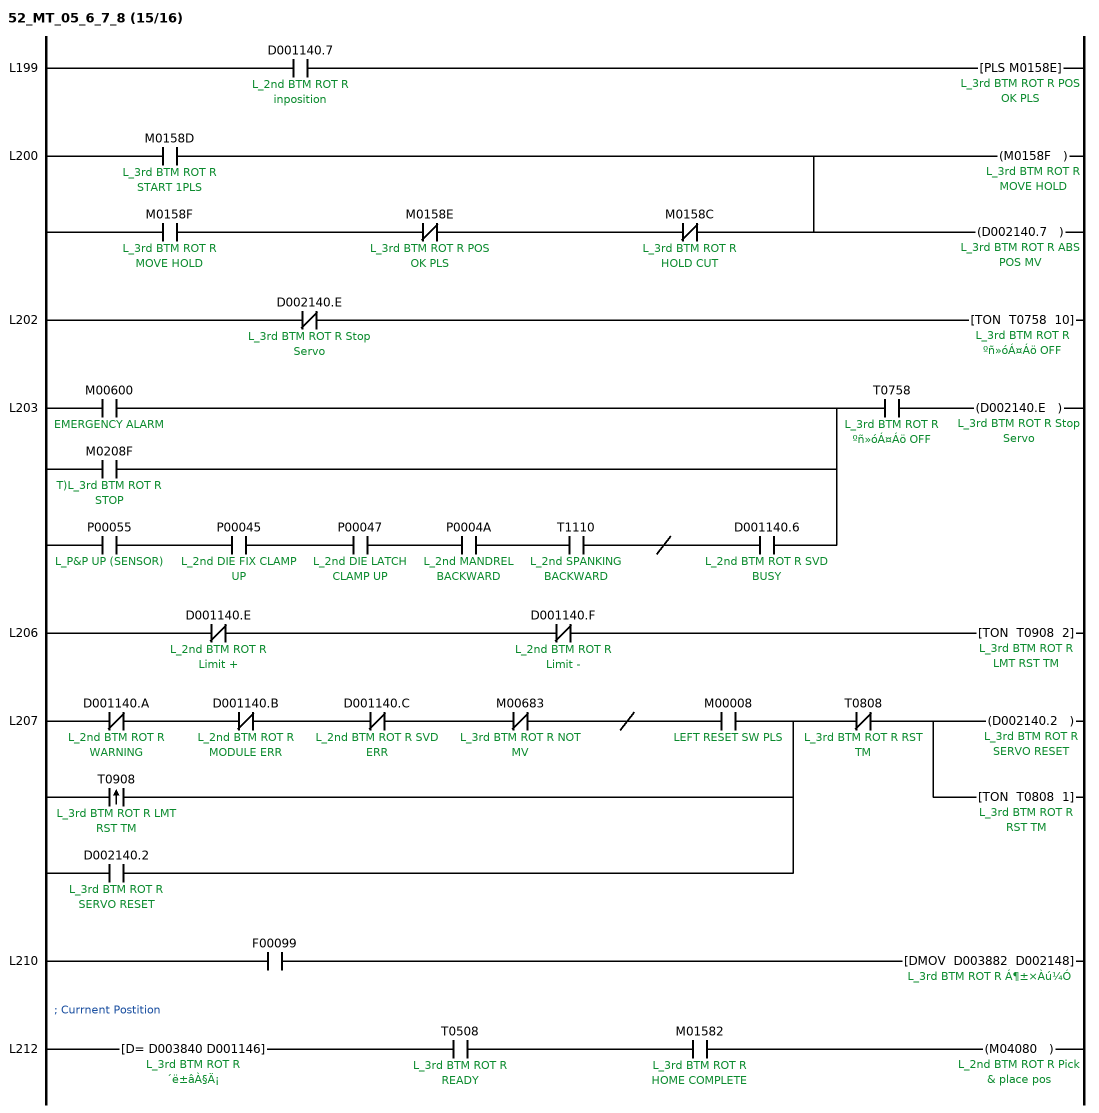
; L199
LOAD      D001140.7	// L_2nd BTM ROT R inposition
OUTP      M0158E	// L_3rd BTM ROT R POS OK PLS
; L200
LOAD      M0158D	// L_3rd BTM ROT R START 1PLS
LOAD      M0158F	// L_3rd BTM ROT R MOVE HOLD
AND NOT   M0158E	// L_3rd BTM ROT R POS OK PLS
AND NOT   M0158C	// L_3rd BTM ROT R HOLD CUT
OR LOAD
OUT       M0158F	// L_3rd BTM ROT R MOVE HOLD
OUT       D002140.7	// L_3rd BTM ROT R ABS POS MV
; L202
LOAD NOT  D002140.E	// L_3rd BTM ROT R Stop Servo
TON       T0758 10	// L_3rd BTM ROT R ºñ»óÁ¤Áö OFF
; L203
LOAD      M00600	// EMERGENCY ALARM
OR        M0208F	// T)L_3rd BTM ROT R STOP
LOAD      P00055	// L_P&P UP (SENSOR)
AND       P00045	// L_2nd DIE FIX CLAMP UP
AND       P00047	// L_2nd DIE LATCH CLAMP UP
AND       P0004A	// L_2nd MANDREL BACKWARD
AND       T1110	// L_2nd SPANKING BACKWARD
NOT
AND       D001140.6	// L_2nd BTM ROT R SVD BUSY
OR LOAD
AND       T0758	// L_3rd BTM ROT R ºñ»óÁ¤Áö OFF
OUT       D002140.E	// L_3rd BTM ROT R Stop Servo
; L206
LOAD NOT  D001140.E	// L_2nd BTM ROT R Limit +
AND NOT   D001140.F	// L_2nd BTM ROT R Limit -
TON       T0908 2	// L_3rd BTM ROT R LMT RST TM
; L207
LOAD NOT  D001140.A	// L_2nd BTM ROT R WARNING
AND NOT   D001140.B	// L_2nd BTM ROT R MODULE ERR
AND NOT   D001140.C	// L_2nd BTM ROT R SVD ERR
AND NOT   M00683	// L_3rd BTM ROT R NOT MV
NOT
AND       M00008	// LEFT RESET SW PLS
ORP       T0908	// L_3rd BTM ROT R LMT RST TM
OR        D002140.2	// L_3rd BTM ROT R SERVO RESET
AND NOT   T0808	// L_3rd BTM ROT R RST TM
OUT       D002140.2	// L_3rd BTM ROT R SERVO RESET
TON       T0808 1	// L_3rd BTM ROT R RST TM
; L210
LOAD      F00099
DMOV      D003882 D002148	// L_3rd BTM ROT R Á¶±×Àú¼Ó
// Currnent Postition
; L212
LOADD=    D003840 D001146	// L_3rd BTM ROT R ´ë±âÀ§Ä¡
AND       T0508	// L_3rd BTM ROT R READY
AND       M01582	// L_3rd BTM ROT R HOME COMPLETE
OUT       M04080	// L_2nd BTM ROT R Pick & place pos

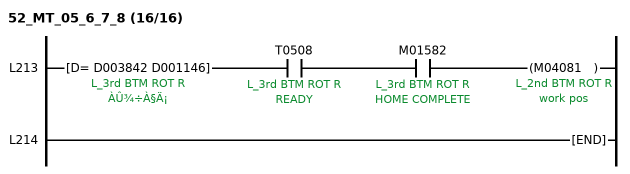
; L213
LOADD=    D003842 D001146	// L_3rd BTM ROT R ÀÛ¾÷À§Ä¡
AND       T0508	// L_3rd BTM ROT R READY
AND       M01582	// L_3rd BTM ROT R HOME COMPLETE
OUT       M04081	// L_2nd BTM ROT R work pos
; L214
END

PROGRAM 53_MT_09_10_11_12 (task: ½ºÄµ ÇÁ·Î±×·¥)

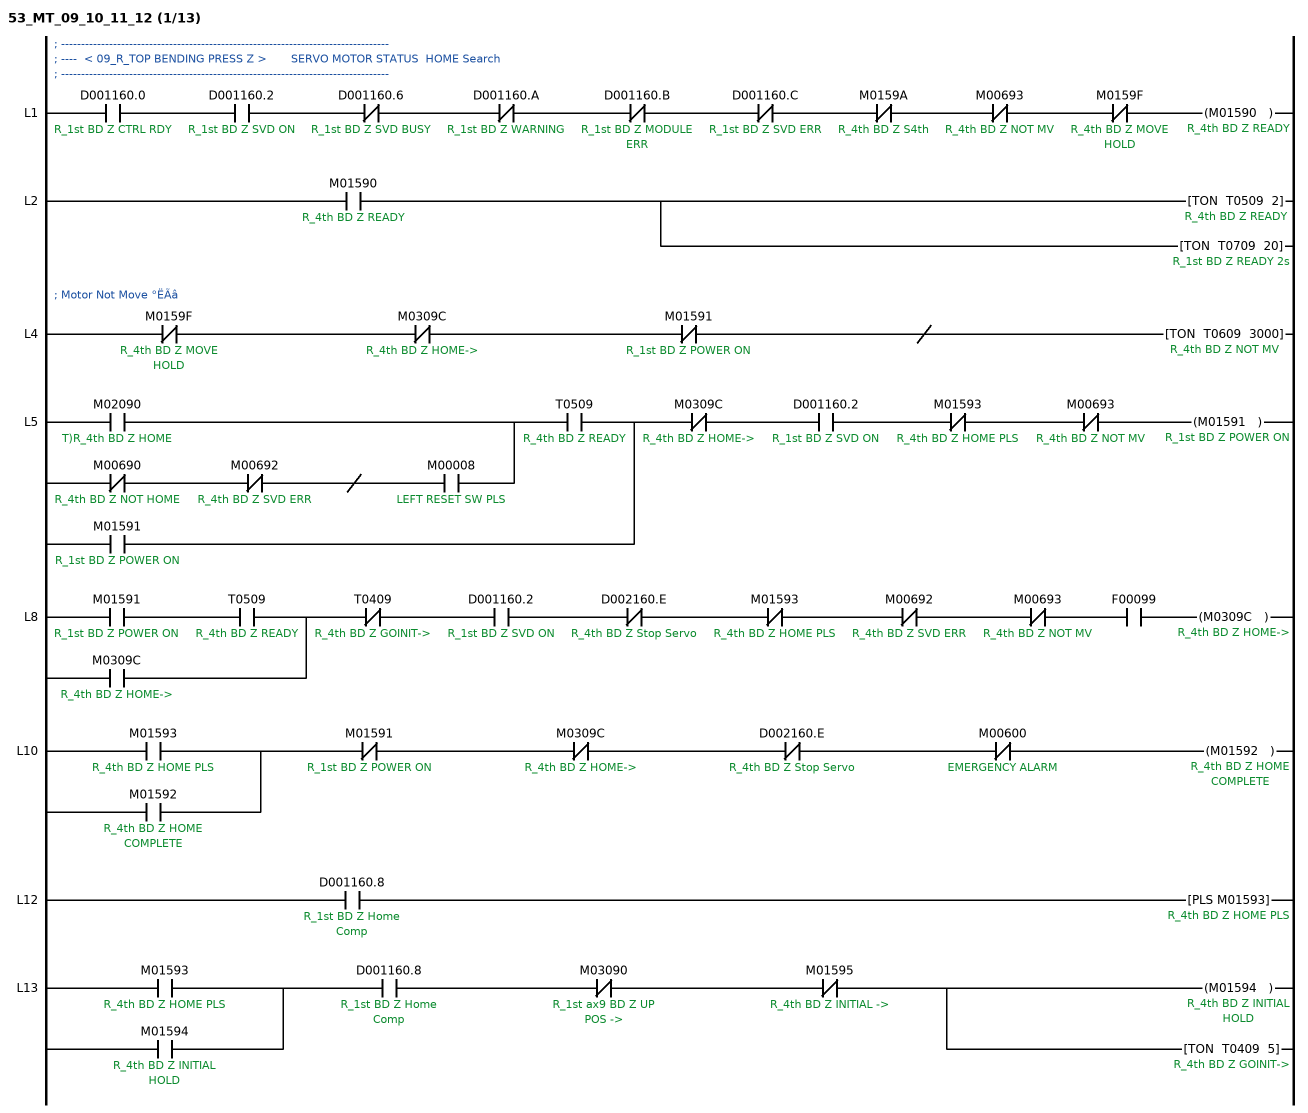
// ----------------------------------------------------------------------------------
// 
// ----  < 09_R_TOP BENDING PRESS Z >       SERVO MOTOR STATUS  HOME Search
// 
// ----------------------------------------------------------------------------------
; L1
LOAD      D001160.0	// R_1st BD Z CTRL RDY
AND       D001160.2	// R_1st BD Z SVD ON
AND NOT   D001160.6	// R_1st BD Z SVD BUSY
AND NOT   D001160.A	// R_1st BD Z WARNING
AND NOT   D001160.B	// R_1st BD Z MODULE ERR
AND NOT   D001160.C	// R_1st BD Z SVD ERR
AND NOT   M0159A	// R_4th BD Z S4th
AND NOT   M00693	// R_4th BD Z NOT MV
AND NOT   M0159F	// R_4th BD Z MOVE HOLD
OUT       M01590	// R_4th BD Z READY
; L2
LOAD      M01590	// R_4th BD Z READY
TON       T0509 2	// R_4th BD Z READY
TON       T0709 20	// R_1st BD Z READY 2s
; L4
LOAD NOT  M0159F	// R_4th BD Z MOVE HOLD
AND NOT   M0309C	// R_4th BD Z HOME->
AND NOT   M01591	// R_1st BD Z POWER ON
NOT
TON       T0609 3000	// R_4th BD Z NOT MV
// output comment: Motor Not Move °ËÃâ
; L5
LOAD      M02090	// T)R_4th BD Z HOME
LOAD NOT  M00690	// R_4th BD Z NOT HOME
AND NOT   M00692	// R_4th BD Z SVD ERR
NOT
AND       M00008	// LEFT RESET SW PLS
OR LOAD
AND       T0509	// R_4th BD Z READY
OR        M01591	// R_1st BD Z POWER ON
AND NOT   M0309C	// R_4th BD Z HOME->
AND       D001160.2	// R_1st BD Z SVD ON
AND NOT   M01593	// R_4th BD Z HOME PLS
AND NOT   M00693	// R_4th BD Z NOT MV
OUT       M01591	// R_1st BD Z POWER ON
; L8
LOAD      M01591	// R_1st BD Z POWER ON
AND       T0509	// R_4th BD Z READY
OR        M0309C	// R_4th BD Z HOME->
AND NOT   T0409	// R_4th BD Z GOINIT->
AND       D001160.2	// R_1st BD Z SVD ON
AND NOT   D002160.E	// R_4th BD Z Stop Servo
AND NOT   M01593	// R_4th BD Z HOME PLS
AND NOT   M00692	// R_4th BD Z SVD ERR
AND NOT   M00693	// R_4th BD Z NOT MV
AND       F00099
OUT       M0309C	// R_4th BD Z HOME->
; L10
LOAD      M01593	// R_4th BD Z HOME PLS
OR        M01592	// R_4th BD Z HOME COMPLETE
AND NOT   M01591	// R_1st BD Z POWER ON
AND NOT   M0309C	// R_4th BD Z HOME->
AND NOT   D002160.E	// R_4th BD Z Stop Servo
AND NOT   M00600	// EMERGENCY ALARM
OUT       M01592	// R_4th BD Z HOME COMPLETE
; L12
LOAD      D001160.8	// R_1st BD Z Home Comp
OUTP      M01593	// R_4th BD Z HOME PLS
; L13
LOAD      M01593	// R_4th BD Z HOME PLS
OR        M01594	// R_4th BD Z INITIAL HOLD
AND       D001160.8	// R_1st BD Z Home Comp
AND NOT   M03090	// R_1st ax9 BD Z UP POS ->
AND NOT   M01595	// R_4th BD Z INITIAL ->
OUT       M01594	// R_4th BD Z INITIAL HOLD
TON       T0409 5	// R_4th BD Z GOINIT->

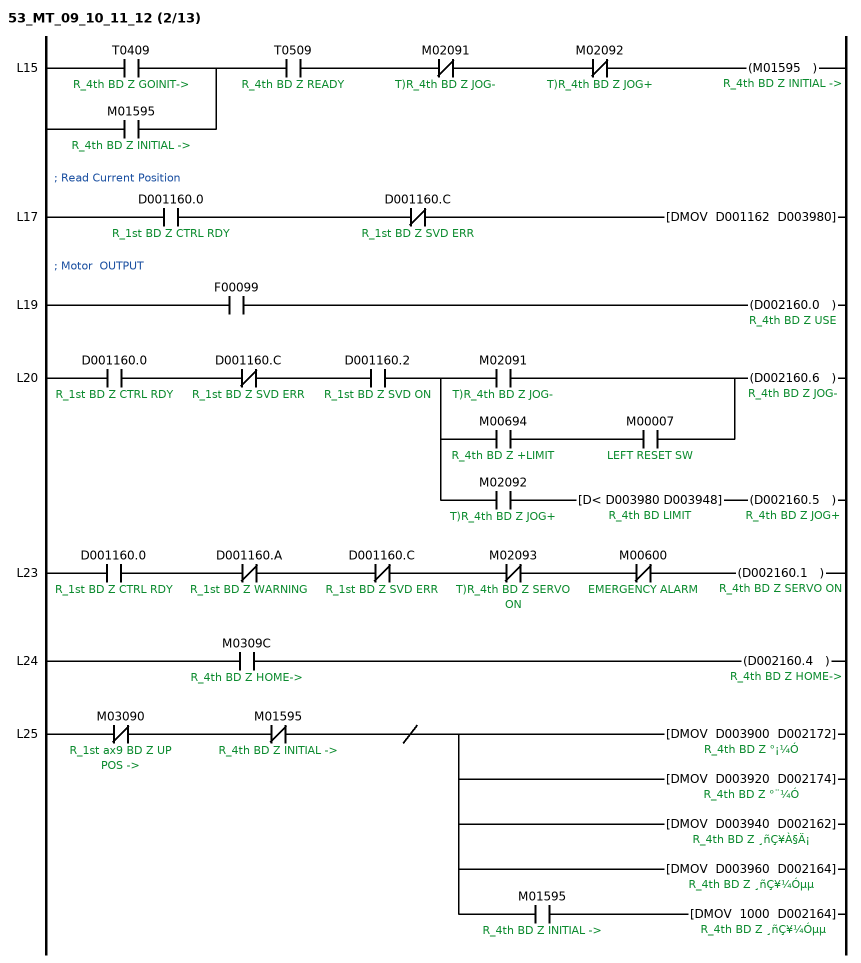
; L15
LOAD      T0409	// R_4th BD Z GOINIT->
OR        M01595	// R_4th BD Z INITIAL ->
AND       T0509	// R_4th BD Z READY
AND NOT   M02091	// T)R_4th BD Z JOG-
AND NOT   M02092	// T)R_4th BD Z JOG+
OUT       M01595	// R_4th BD Z INITIAL ->
; L17
LOAD      D001160.0	// R_1st BD Z CTRL RDY
AND NOT   D001160.C	// R_1st BD Z SVD ERR
DMOV      D001162 D003980
// output comment: Read Current Position
//  Motor  OUTPUT
; L19
LOAD      F00099
OUT       D002160.0	// R_4th BD Z USE
; L20
LOAD      D001160.0	// R_1st BD Z CTRL RDY
AND NOT   D001160.C	// R_1st BD Z SVD ERR
AND       D001160.2	// R_1st BD Z SVD ON
MPUSH
LOAD      M02091	// T)R_4th BD Z JOG-
LOAD      M00694	// R_4th BD Z +LIMIT
AND       M00007	// LEFT RESET SW
OR LOAD
AND LOAD
OUT       D002160.6	// R_4th BD Z JOG-
MPOP
AND       M02092	// T)R_4th BD Z JOG+
ANDD<     D003980 D003948	// R_4th BD LIMIT
OUT       D002160.5	// R_4th BD Z JOG+
; L23
LOAD      D001160.0	// R_1st BD Z CTRL RDY
AND NOT   D001160.A	// R_1st BD Z WARNING
AND NOT   D001160.C	// R_1st BD Z SVD ERR
AND NOT   M02093	// T)R_4th BD Z SERVO ON
AND NOT   M00600	// EMERGENCY ALARM
OUT       D002160.1	// R_4th BD Z SERVO ON
; L24
LOAD      M0309C	// R_4th BD Z HOME->
OUT       D002160.4	// R_4th BD Z HOME->
; L25
LOAD NOT  M03090	// R_1st ax9 BD Z UP POS ->
AND NOT   M01595	// R_4th BD Z INITIAL ->
NOT
DMOV      D003900 D002172	// R_4th BD Z °¡¼Ó
DMOV      D003920 D002174	// R_4th BD Z °¨¼Ó
DMOV      D003940 D002162	// R_4th BD Z ¸ñÇ¥À§Ä¡
DMOV      D003960 D002164	// R_4th BD Z ¸ñÇ¥¼Óµµ
AND       M01595	// R_4th BD Z INITIAL ->
DMOV      1000 D002164	// R_4th BD Z ¸ñÇ¥¼Óµµ

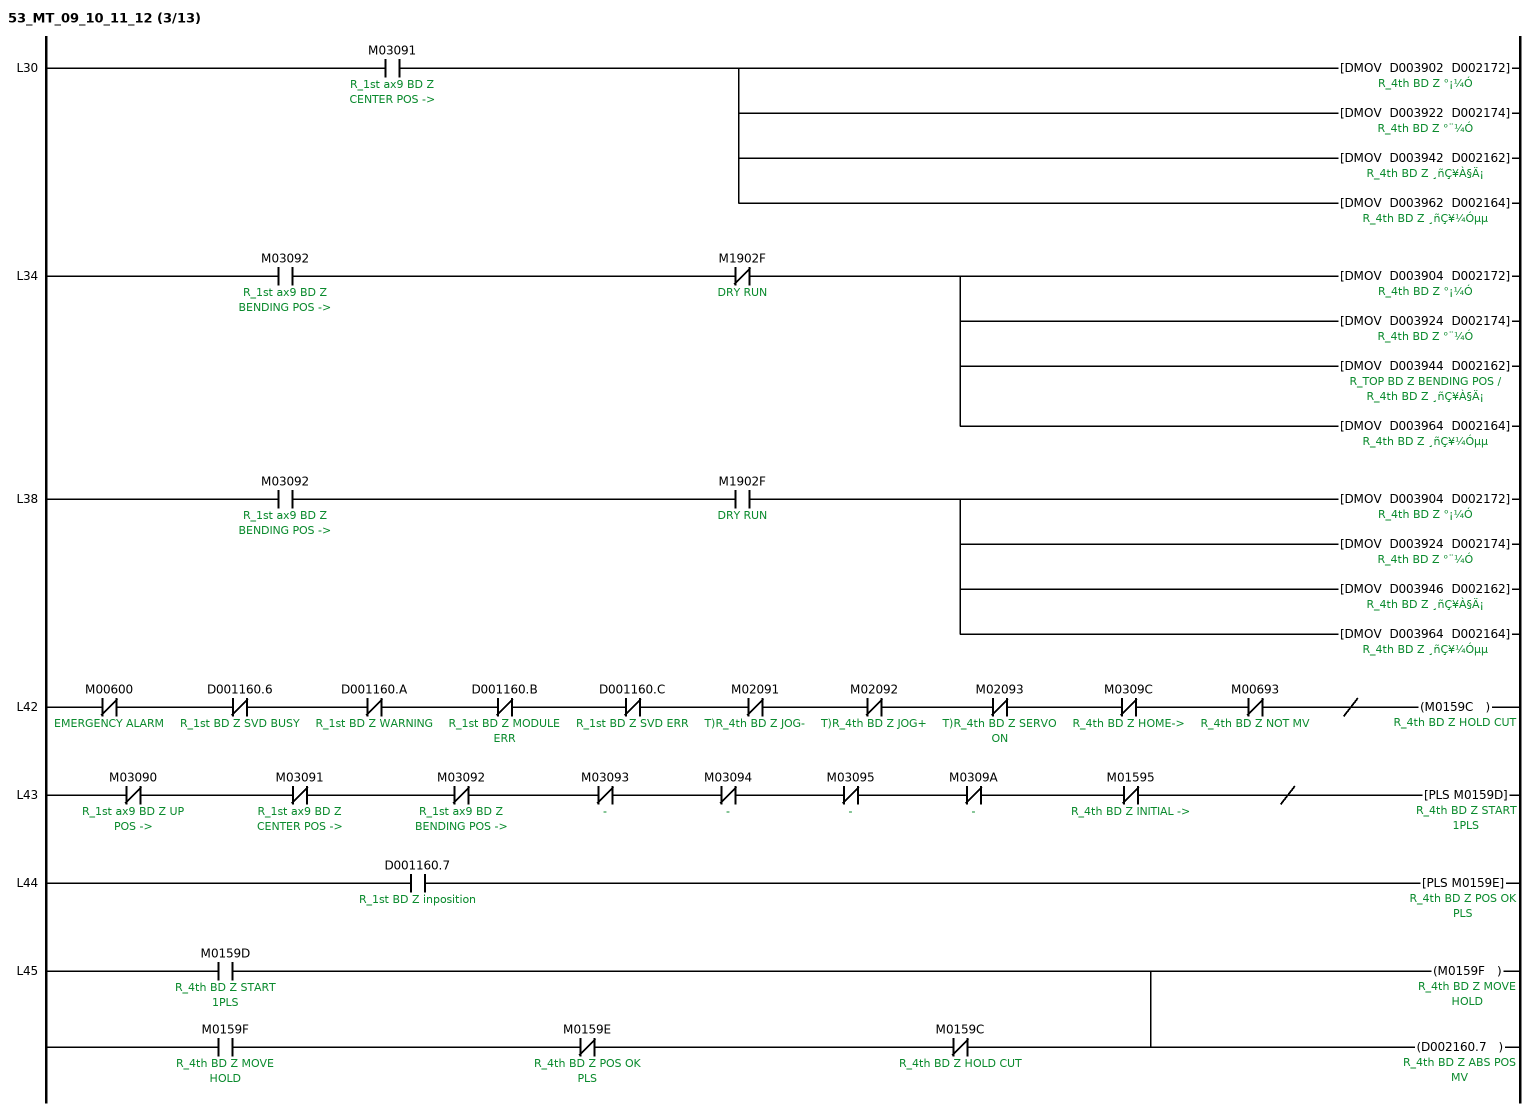
; L30
LOAD      M03091	// R_1st ax9 BD Z CENTER POS ->
DMOV      D003902 D002172	// R_4th BD Z °¡¼Ó
DMOV      D003922 D002174	// R_4th BD Z °¨¼Ó
DMOV      D003942 D002162	// R_4th BD Z ¸ñÇ¥À§Ä¡
DMOV      D003962 D002164	// R_4th BD Z ¸ñÇ¥¼Óµµ
; L34
LOAD      M03092	// R_1st ax9 BD Z BENDING POS ->
AND NOT   M1902F	// DRY RUN
DMOV      D003904 D002172	// R_4th BD Z °¡¼Ó
DMOV      D003924 D002174	// R_4th BD Z °¨¼Ó
DMOV      D003944 D002162	// R_TOP BD Z BENDING POS / R_4th BD Z ¸ñÇ¥À§Ä¡
DMOV      D003964 D002164	// R_4th BD Z ¸ñÇ¥¼Óµµ
; L38
LOAD      M03092	// R_1st ax9 BD Z BENDING POS ->
AND       M1902F	// DRY RUN
DMOV      D003904 D002172	// R_4th BD Z °¡¼Ó
DMOV      D003924 D002174	// R_4th BD Z °¨¼Ó
DMOV      D003946 D002162	// R_4th BD Z ¸ñÇ¥À§Ä¡
DMOV      D003964 D002164	// R_4th BD Z ¸ñÇ¥¼Óµµ
; L42
LOAD NOT  M00600	// EMERGENCY ALARM
AND NOT   D001160.6	// R_1st BD Z SVD BUSY
AND NOT   D001160.A	// R_1st BD Z WARNING
AND NOT   D001160.B	// R_1st BD Z MODULE ERR
AND NOT   D001160.C	// R_1st BD Z SVD ERR
AND NOT   M02091	// T)R_4th BD Z JOG-
AND NOT   M02092	// T)R_4th BD Z JOG+
AND NOT   M02093	// T)R_4th BD Z SERVO ON
AND NOT   M0309C	// R_4th BD Z HOME->
AND NOT   M00693	// R_4th BD Z NOT MV
NOT
OUT       M0159C	// R_4th BD Z HOLD CUT
; L43
LOAD NOT  M03090	// R_1st ax9 BD Z UP POS ->
AND NOT   M03091	// R_1st ax9 BD Z CENTER POS ->
AND NOT   M03092	// R_1st ax9 BD Z BENDING POS ->
AND NOT   M03093	// -
AND NOT   M03094	// -
AND NOT   M03095	// -
AND NOT   M0309A	// -
AND NOT   M01595	// R_4th BD Z INITIAL ->
NOT
OUTP      M0159D	// R_4th BD Z START 1PLS
; L44
LOAD      D001160.7	// R_1st BD Z inposition
OUTP      M0159E	// R_4th BD Z POS OK PLS
; L45
LOAD      M0159D	// R_4th BD Z START 1PLS
LOAD      M0159F	// R_4th BD Z MOVE HOLD
AND NOT   M0159E	// R_4th BD Z POS OK PLS
AND NOT   M0159C	// R_4th BD Z HOLD CUT
OR LOAD
OUT       M0159F	// R_4th BD Z MOVE HOLD
OUT       D002160.7	// R_4th BD Z ABS POS MV

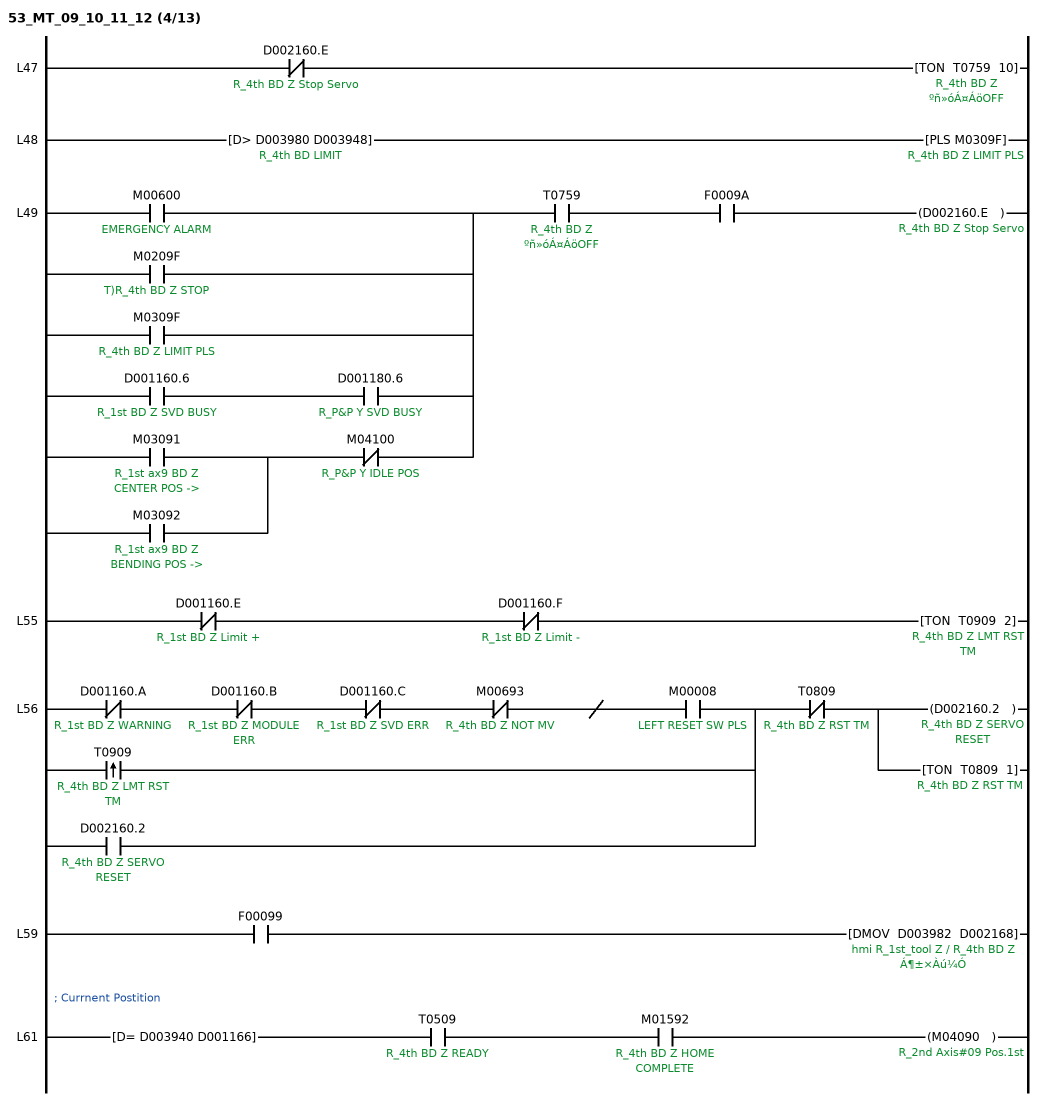
; L47
LOAD NOT  D002160.E	// R_4th BD Z Stop Servo
TON       T0759 10	// R_4th BD Z ºñ»óÁ¤ÁöOFF
; L48
LOADD>    D003980 D003948	// R_4th BD LIMIT
OUTP      M0309F	// R_4th BD Z LIMIT PLS
; L49
LOAD      M00600	// EMERGENCY ALARM
OR        M0209F	// T)R_4th BD Z STOP
OR        M0309F	// R_4th BD Z LIMIT PLS
LOAD      D001160.6	// R_1st BD Z SVD BUSY
AND       D001180.6	// R_P&P Y SVD BUSY
OR LOAD
LOAD      M03091	// R_1st ax9 BD Z CENTER POS ->
OR        M03092	// R_1st ax9 BD Z BENDING POS ->
AND NOT   M04100	// R_P&P Y IDLE POS
OR LOAD
AND       T0759	// R_4th BD Z ºñ»óÁ¤ÁöOFF
AND       F0009A
OUT       D002160.E	// R_4th BD Z Stop Servo
; L55
LOAD NOT  D001160.E	// R_1st BD Z Limit +
AND NOT   D001160.F	// R_1st BD Z Limit -
TON       T0909 2	// R_4th BD Z LMT RST TM
; L56
LOAD NOT  D001160.A	// R_1st BD Z WARNING
AND NOT   D001160.B	// R_1st BD Z MODULE ERR
AND NOT   D001160.C	// R_1st BD Z SVD ERR
AND NOT   M00693	// R_4th BD Z NOT MV
NOT
AND       M00008	// LEFT RESET SW PLS
ORP       T0909	// R_4th BD Z LMT RST TM
OR        D002160.2	// R_4th BD Z SERVO RESET
AND NOT   T0809	// R_4th BD Z RST TM
OUT       D002160.2	// R_4th BD Z SERVO RESET
TON       T0809 1	// R_4th BD Z RST TM
; L59
LOAD      F00099
DMOV      D003982 D002168	// hmi R_1st_tool Z / R_4th BD Z Á¶±×Àú¼Ó
// Currnent Postition
; L61
LOADD=    D003940 D001166
AND       T0509	// R_4th BD Z READY
AND       M01592	// R_4th BD Z HOME COMPLETE
OUT       M04090	// R_2nd Axis#09 Pos.1st

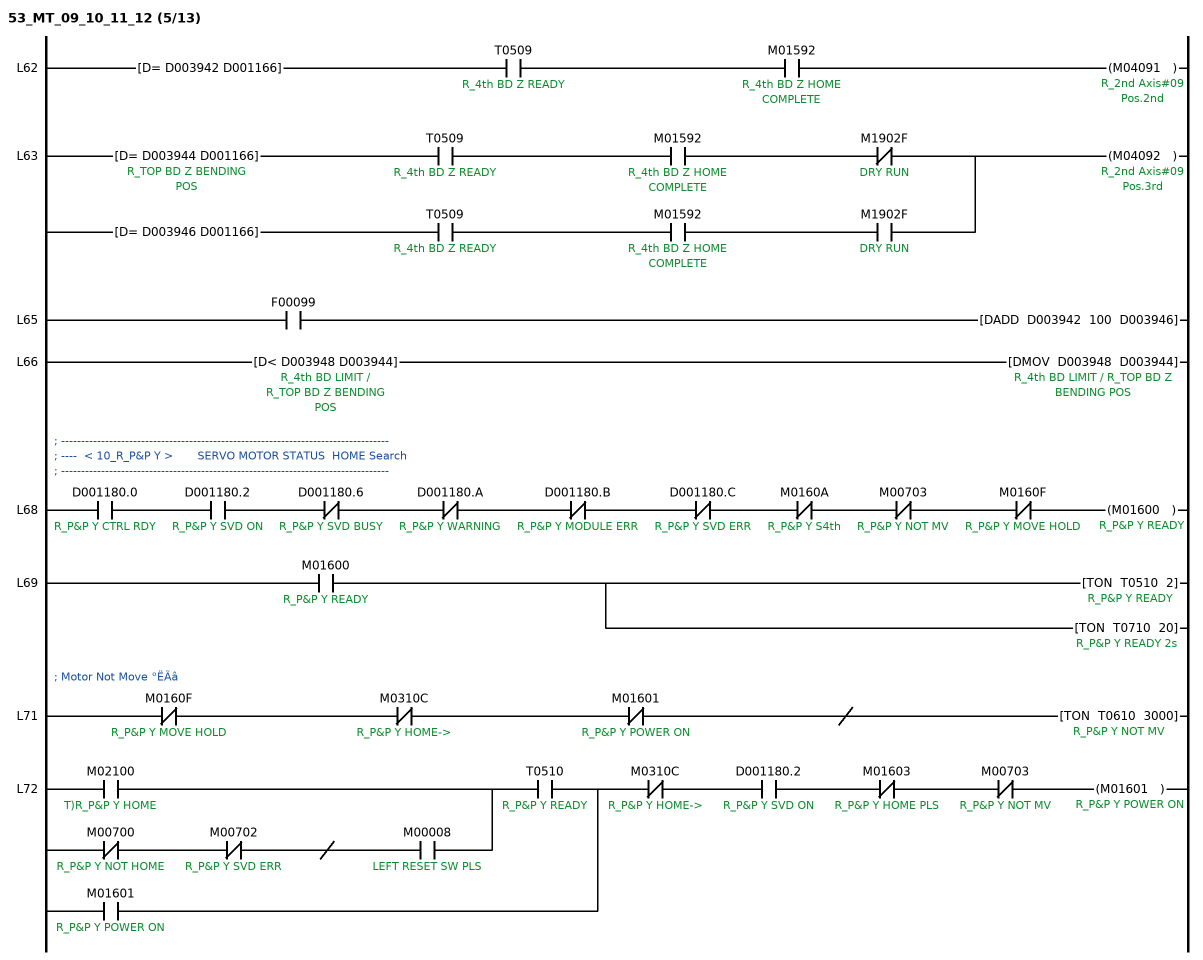
; L62
LOADD=    D003942 D001166
AND       T0509	// R_4th BD Z READY
AND       M01592	// R_4th BD Z HOME COMPLETE
OUT       M04091	// R_2nd Axis#09 Pos.2nd
; L63
LOADD=    D003944 D001166	// R_TOP BD Z BENDING POS
AND       T0509	// R_4th BD Z READY
AND       M01592	// R_4th BD Z HOME COMPLETE
AND NOT   M1902F	// DRY RUN
LOADD=    D003946 D001166
AND       T0509	// R_4th BD Z READY
AND       M01592	// R_4th BD Z HOME COMPLETE
AND       M1902F	// DRY RUN
OR LOAD
OUT       M04092	// R_2nd Axis#09 Pos.3rd
; L65
LOAD      F00099
DADD      D003942 100 D003946
; L66
LOADD<    D003948 D003944	// R_4th BD LIMIT / R_TOP BD Z BENDING POS
DMOV      D003948 D003944	// R_4th BD LIMIT / R_TOP BD Z BENDING POS
// ----------------------------------------------------------------------------------
// 
// ----  < 10_R_P&P Y >       SERVO MOTOR STATUS  HOME Search
// 
// ----------------------------------------------------------------------------------
; L68
LOAD      D001180.0	// R_P&P Y CTRL RDY
AND       D001180.2	// R_P&P Y SVD ON
AND NOT   D001180.6	// R_P&P Y SVD BUSY
AND NOT   D001180.A	// R_P&P Y WARNING
AND NOT   D001180.B	// R_P&P Y MODULE ERR
AND NOT   D001180.C	// R_P&P Y SVD ERR
AND NOT   M0160A	// R_P&P Y S4th
AND NOT   M00703	// R_P&P Y NOT MV
AND NOT   M0160F	// R_P&P Y MOVE HOLD
OUT       M01600	// R_P&P Y READY
; L69
LOAD      M01600	// R_P&P Y READY
TON       T0510 2	// R_P&P Y READY
TON       T0710 20	// R_P&P Y READY 2s
; L71
LOAD NOT  M0160F	// R_P&P Y MOVE HOLD
AND NOT   M0310C	// R_P&P Y HOME->
AND NOT   M01601	// R_P&P Y POWER ON
NOT
TON       T0610 3000	// R_P&P Y NOT MV
// output comment: Motor Not Move °ËÃâ
; L72
LOAD      M02100	// T)R_P&P Y HOME
LOAD NOT  M00700	// R_P&P Y NOT HOME
AND NOT   M00702	// R_P&P Y SVD ERR
NOT
AND       M00008	// LEFT RESET SW PLS
OR LOAD
AND       T0510	// R_P&P Y READY
OR        M01601	// R_P&P Y POWER ON
AND NOT   M0310C	// R_P&P Y HOME->
AND       D001180.2	// R_P&P Y SVD ON
AND NOT   M01603	// R_P&P Y HOME PLS
AND NOT   M00703	// R_P&P Y NOT MV
OUT       M01601	// R_P&P Y POWER ON

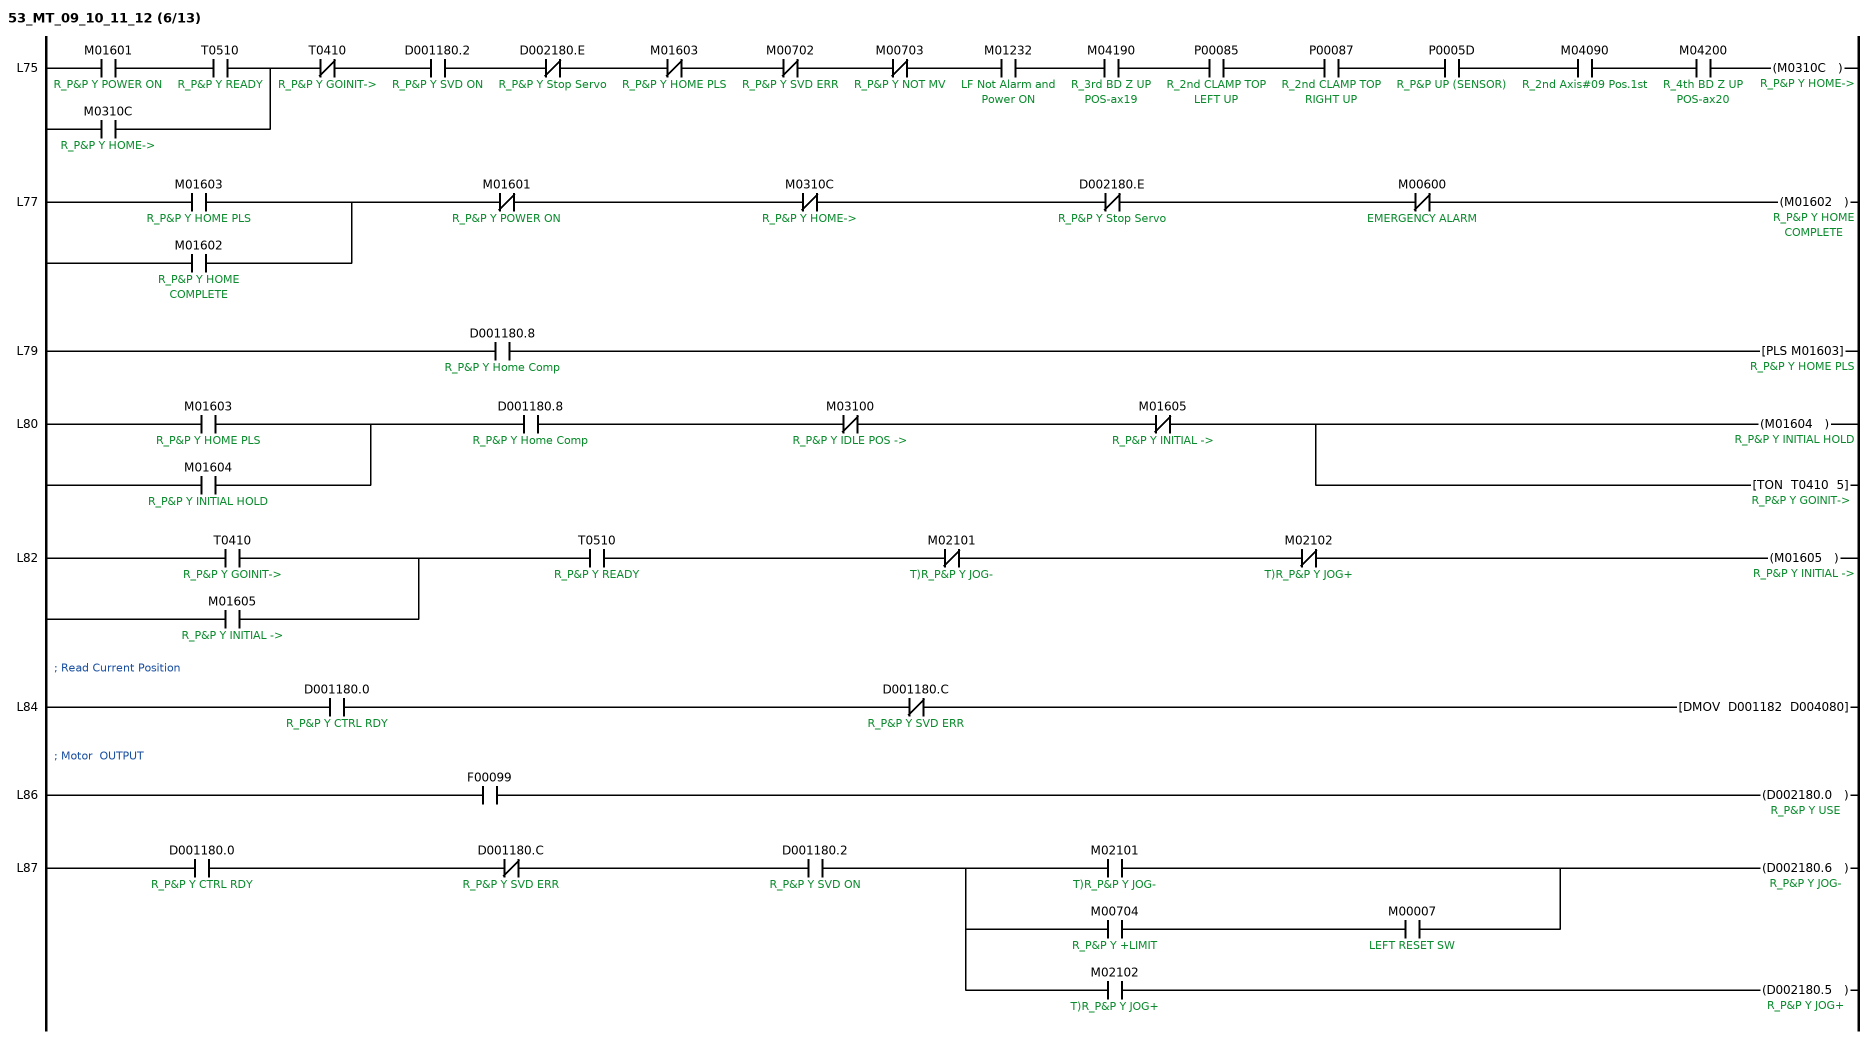
; L75
LOAD      M01601	// R_P&P Y POWER ON
AND       T0510	// R_P&P Y READY
OR        M0310C	// R_P&P Y HOME->
AND NOT   T0410	// R_P&P Y GOINIT->
AND       D001180.2	// R_P&P Y SVD ON
AND NOT   D002180.E	// R_P&P Y Stop Servo
AND NOT   M01603	// R_P&P Y HOME PLS
AND NOT   M00702	// R_P&P Y SVD ERR
AND NOT   M00703	// R_P&P Y NOT MV
AND       M01232	// LF Not Alarm and Power ON
AND       M04190	// R_3rd BD Z UP POS-ax19
AND       P00085	// R_2nd CLAMP TOP LEFT UP
AND       P00087	// R_2nd CLAMP TOP RIGHT UP
AND       P0005D	// R_P&P UP (SENSOR)
AND       M04090	// R_2nd Axis#09 Pos.1st
AND       M04200	// R_4th BD Z UP POS-ax20
OUT       M0310C	// R_P&P Y HOME->
; L77
LOAD      M01603	// R_P&P Y HOME PLS
OR        M01602	// R_P&P Y HOME COMPLETE
AND NOT   M01601	// R_P&P Y POWER ON
AND NOT   M0310C	// R_P&P Y HOME->
AND NOT   D002180.E	// R_P&P Y Stop Servo
AND NOT   M00600	// EMERGENCY ALARM
OUT       M01602	// R_P&P Y HOME COMPLETE
; L79
LOAD      D001180.8	// R_P&P Y Home Comp
OUTP      M01603	// R_P&P Y HOME PLS
; L80
LOAD      M01603	// R_P&P Y HOME PLS
OR        M01604	// R_P&P Y INITIAL HOLD
AND       D001180.8	// R_P&P Y Home Comp
AND NOT   M03100	// R_P&P Y IDLE POS ->
AND NOT   M01605	// R_P&P Y INITIAL ->
OUT       M01604	// R_P&P Y INITIAL HOLD
TON       T0410 5	// R_P&P Y GOINIT->
; L82
LOAD      T0410	// R_P&P Y GOINIT->
OR        M01605	// R_P&P Y INITIAL ->
AND       T0510	// R_P&P Y READY
AND NOT   M02101	// T)R_P&P Y JOG-
AND NOT   M02102	// T)R_P&P Y JOG+
OUT       M01605	// R_P&P Y INITIAL ->
; L84
LOAD      D001180.0	// R_P&P Y CTRL RDY
AND NOT   D001180.C	// R_P&P Y SVD ERR
DMOV      D001182 D004080
// output comment: Read Current Position
//  Motor  OUTPUT
; L86
LOAD      F00099
OUT       D002180.0	// R_P&P Y USE
; L87
LOAD      D001180.0	// R_P&P Y CTRL RDY
AND NOT   D001180.C	// R_P&P Y SVD ERR
AND       D001180.2	// R_P&P Y SVD ON
MPUSH
LOAD      M02101	// T)R_P&P Y JOG-
LOAD      M00704	// R_P&P Y +LIMIT
AND       M00007	// LEFT RESET SW
OR LOAD
AND LOAD
OUT       D002180.6	// R_P&P Y JOG-
MPOP
AND       M02102	// T)R_P&P Y JOG+
OUT       D002180.5	// R_P&P Y JOG+

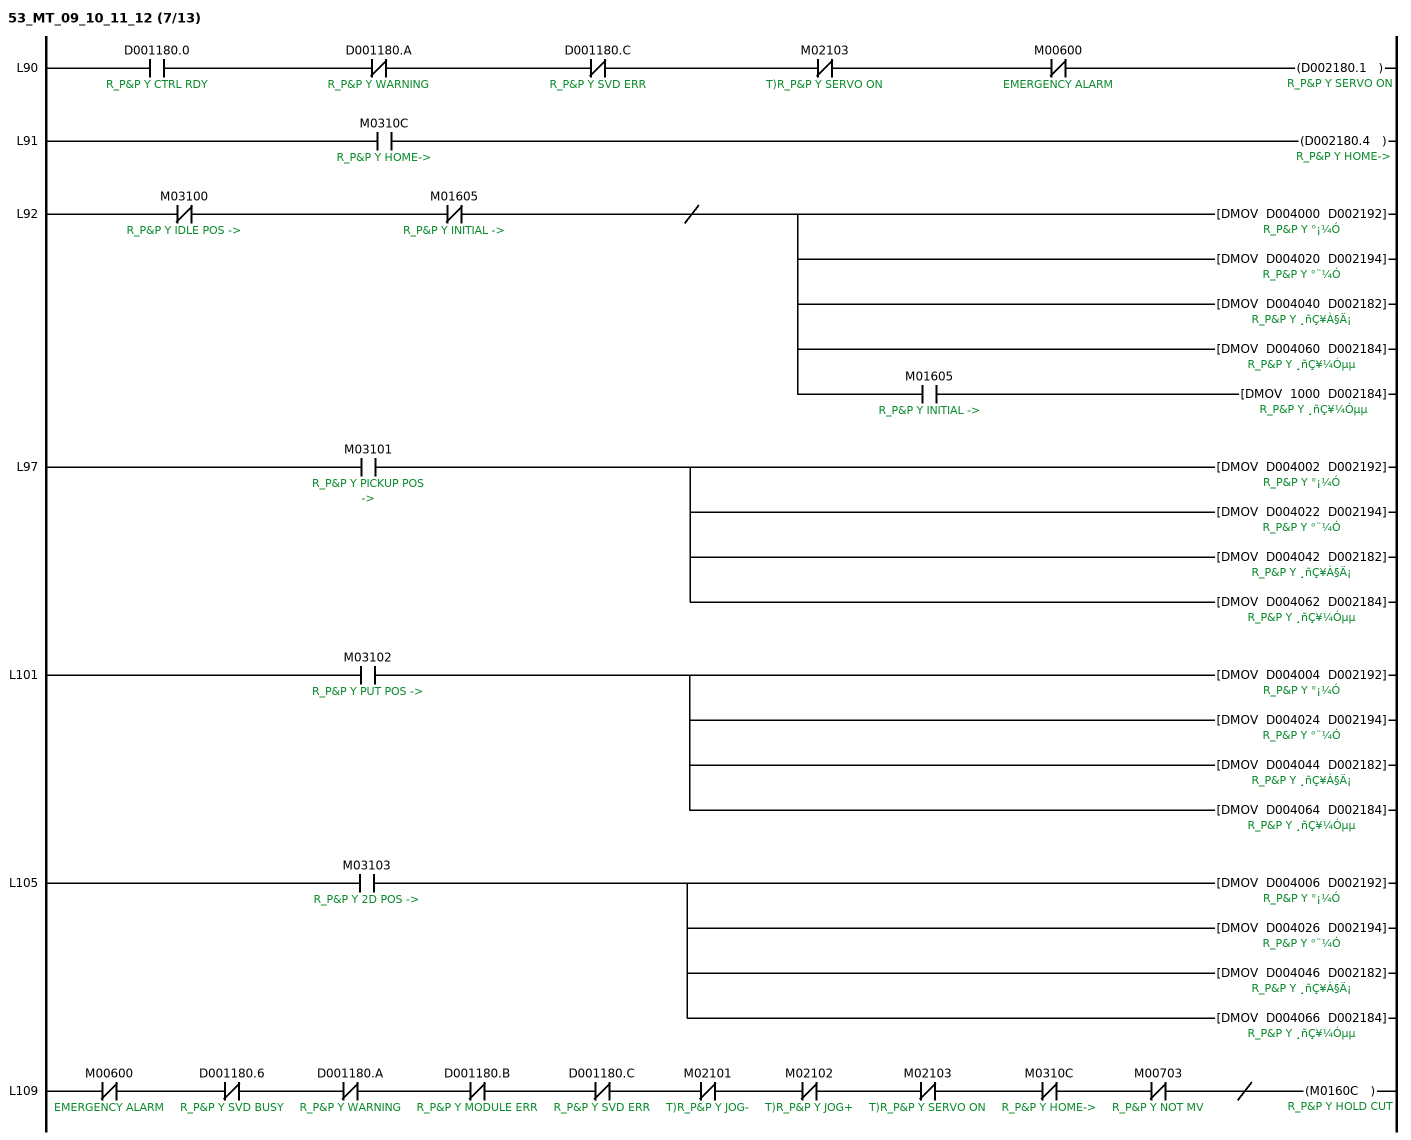
; L90
LOAD      D001180.0	// R_P&P Y CTRL RDY
AND NOT   D001180.A	// R_P&P Y WARNING
AND NOT   D001180.C	// R_P&P Y SVD ERR
AND NOT   M02103	// T)R_P&P Y SERVO ON
AND NOT   M00600	// EMERGENCY ALARM
OUT       D002180.1	// R_P&P Y SERVO ON
; L91
LOAD      M0310C	// R_P&P Y HOME->
OUT       D002180.4	// R_P&P Y HOME->
; L92
LOAD NOT  M03100	// R_P&P Y IDLE POS ->
AND NOT   M01605	// R_P&P Y INITIAL ->
NOT
DMOV      D004000 D002192	// R_P&P Y °¡¼Ó
DMOV      D004020 D002194	// R_P&P Y °¨¼Ó
DMOV      D004040 D002182	// R_P&P Y ¸ñÇ¥À§Ä¡
DMOV      D004060 D002184	// R_P&P Y ¸ñÇ¥¼Óµµ
AND       M01605	// R_P&P Y INITIAL ->
DMOV      1000 D002184	// R_P&P Y ¸ñÇ¥¼Óµµ
; L97
LOAD      M03101	// R_P&P Y PICKUP POS ->
DMOV      D004002 D002192	// R_P&P Y °¡¼Ó
DMOV      D004022 D002194	// R_P&P Y °¨¼Ó
DMOV      D004042 D002182	// R_P&P Y ¸ñÇ¥À§Ä¡
DMOV      D004062 D002184	// R_P&P Y ¸ñÇ¥¼Óµµ
; L101
LOAD      M03102	// R_P&P Y PUT POS ->
DMOV      D004004 D002192	// R_P&P Y °¡¼Ó
DMOV      D004024 D002194	// R_P&P Y °¨¼Ó
DMOV      D004044 D002182	// R_P&P Y ¸ñÇ¥À§Ä¡
DMOV      D004064 D002184	// R_P&P Y ¸ñÇ¥¼Óµµ
; L105
LOAD      M03103	// R_P&P Y 2D POS ->
DMOV      D004006 D002192	// R_P&P Y °¡¼Ó
DMOV      D004026 D002194	// R_P&P Y °¨¼Ó
DMOV      D004046 D002182	// R_P&P Y ¸ñÇ¥À§Ä¡
DMOV      D004066 D002184	// R_P&P Y ¸ñÇ¥¼Óµµ
; L109
LOAD NOT  M00600	// EMERGENCY ALARM
AND NOT   D001180.6	// R_P&P Y SVD BUSY
AND NOT   D001180.A	// R_P&P Y WARNING
AND NOT   D001180.B	// R_P&P Y MODULE ERR
AND NOT   D001180.C	// R_P&P Y SVD ERR
AND NOT   M02101	// T)R_P&P Y JOG-
AND NOT   M02102	// T)R_P&P Y JOG+
AND NOT   M02103	// T)R_P&P Y SERVO ON
AND NOT   M0310C	// R_P&P Y HOME->
AND NOT   M00703	// R_P&P Y NOT MV
NOT
OUT       M0160C	// R_P&P Y HOLD CUT

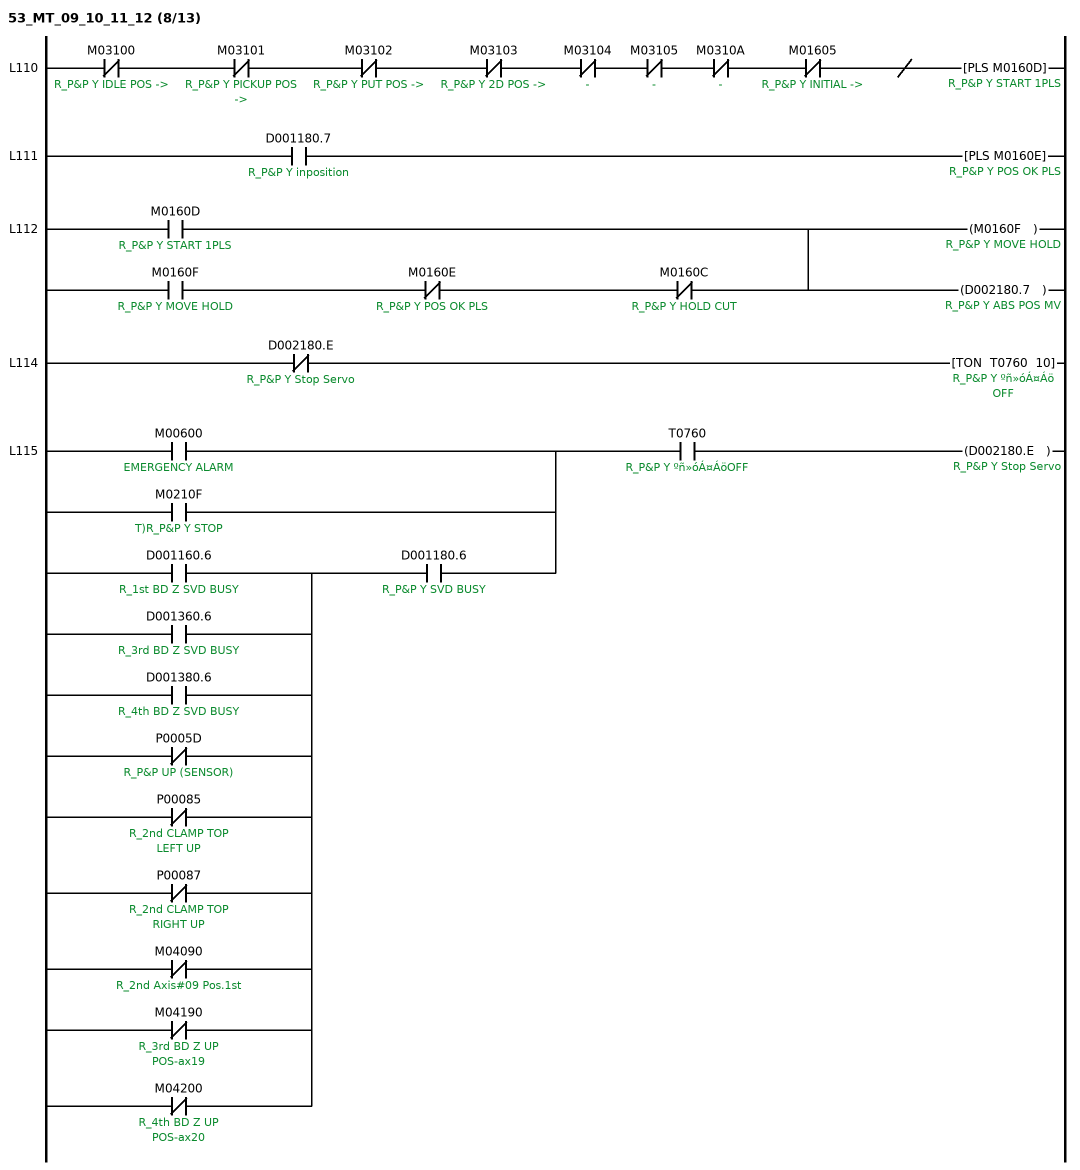
; L110
LOAD NOT  M03100	// R_P&P Y IDLE POS ->
AND NOT   M03101	// R_P&P Y PICKUP POS ->
AND NOT   M03102	// R_P&P Y PUT POS ->
AND NOT   M03103	// R_P&P Y 2D POS ->
AND NOT   M03104	// -
AND NOT   M03105	// -
AND NOT   M0310A	// -
AND NOT   M01605	// R_P&P Y INITIAL ->
NOT
OUTP      M0160D	// R_P&P Y START 1PLS
; L111
LOAD      D001180.7	// R_P&P Y inposition
OUTP      M0160E	// R_P&P Y POS OK PLS
; L112
LOAD      M0160D	// R_P&P Y START 1PLS
LOAD      M0160F	// R_P&P Y MOVE HOLD
AND NOT   M0160E	// R_P&P Y POS OK PLS
AND NOT   M0160C	// R_P&P Y HOLD CUT
OR LOAD
OUT       M0160F	// R_P&P Y MOVE HOLD
OUT       D002180.7	// R_P&P Y ABS POS MV
; L114
LOAD NOT  D002180.E	// R_P&P Y Stop Servo
TON       T0760 10	// R_P&P Y ºñ»óÁ¤ÁöOFF
; L115
LOAD      M00600	// EMERGENCY ALARM
OR        M0210F	// T)R_P&P Y STOP
LOAD      D001160.6	// R_1st BD Z SVD BUSY
OR        D001360.6	// R_3rd BD Z SVD BUSY
OR        D001380.6	// R_4th BD Z SVD BUSY
OR NOT    P0005D	// R_P&P UP (SENSOR)
OR NOT    P00085	// R_2nd CLAMP TOP LEFT UP
OR NOT    P00087	// R_2nd CLAMP TOP RIGHT UP
OR NOT    M04090	// R_2nd Axis#09 Pos.1st
OR NOT    M04190	// R_3rd BD Z UP POS-ax19
OR NOT    M04200	// R_4th BD Z UP POS-ax20
AND       D001180.6	// R_P&P Y SVD BUSY
OR LOAD
AND       T0760	// R_P&P Y ºñ»óÁ¤ÁöOFF
OUT       D002180.E	// R_P&P Y Stop Servo

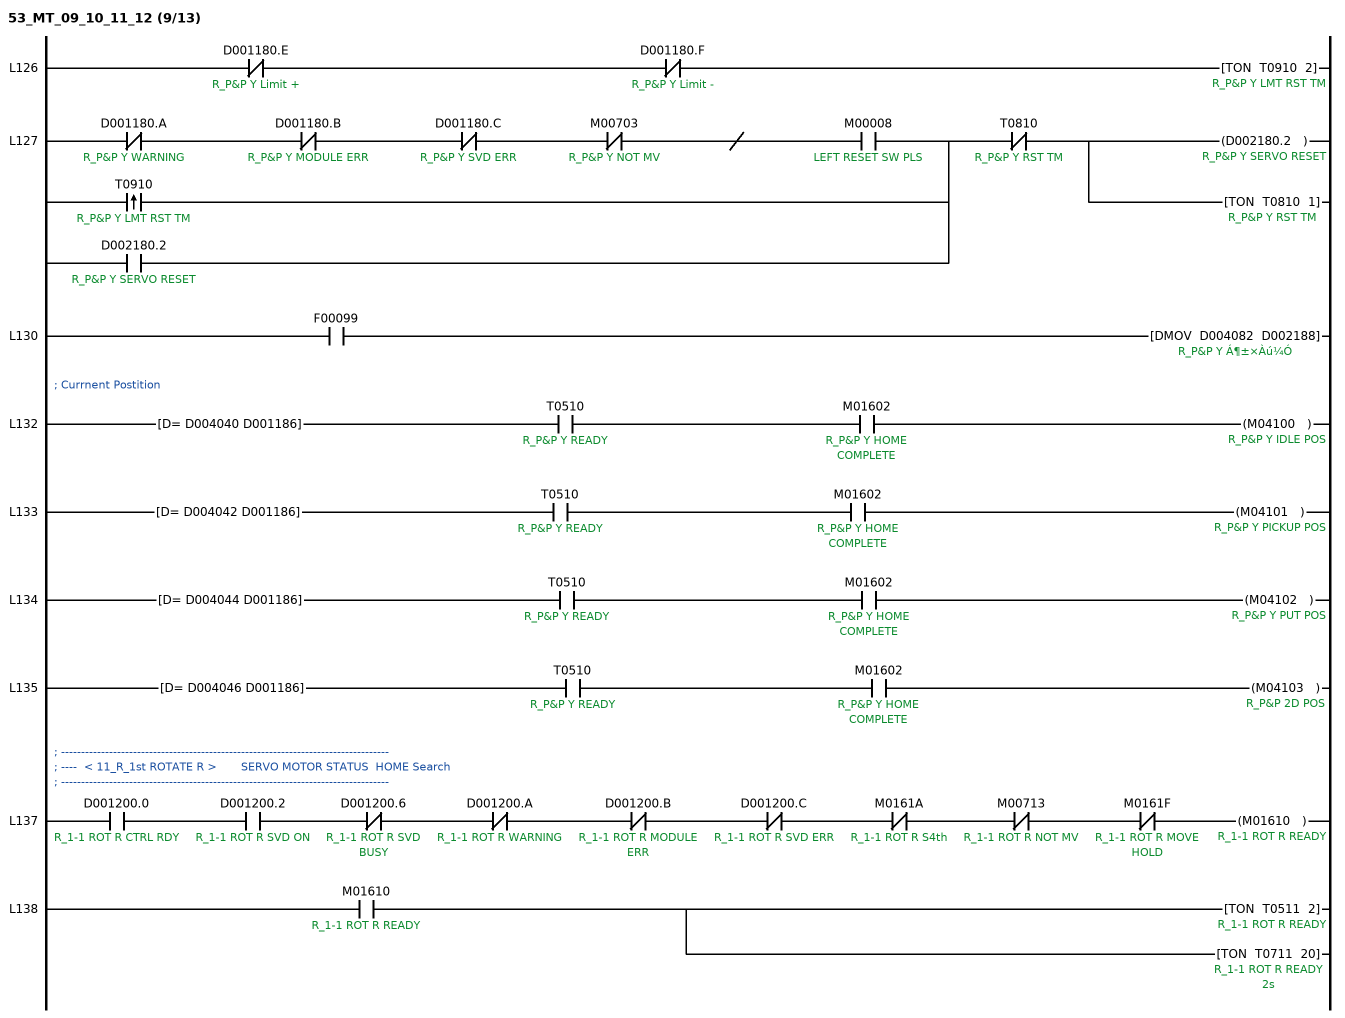
; L126
LOAD NOT  D001180.E	// R_P&P Y Limit +
AND NOT   D001180.F	// R_P&P Y Limit -
TON       T0910 2	// R_P&P Y LMT RST TM
; L127
LOAD NOT  D001180.A	// R_P&P Y WARNING
AND NOT   D001180.B	// R_P&P Y MODULE ERR
AND NOT   D001180.C	// R_P&P Y SVD ERR
AND NOT   M00703	// R_P&P Y NOT MV
NOT
AND       M00008	// LEFT RESET SW PLS
ORP       T0910	// R_P&P Y LMT RST TM
OR        D002180.2	// R_P&P Y SERVO RESET
AND NOT   T0810	// R_P&P Y RST TM
OUT       D002180.2	// R_P&P Y SERVO RESET
TON       T0810 1	// R_P&P Y RST TM
; L130
LOAD      F00099
DMOV      D004082 D002188	// R_P&P Y Á¶±×Àú¼Ó
// Currnent Postition
; L132
LOADD=    D004040 D001186
AND       T0510	// R_P&P Y READY
AND       M01602	// R_P&P Y HOME COMPLETE
OUT       M04100	// R_P&P Y IDLE POS
; L133
LOADD=    D004042 D001186
AND       T0510	// R_P&P Y READY
AND       M01602	// R_P&P Y HOME COMPLETE
OUT       M04101	// R_P&P Y PICKUP POS
; L134
LOADD=    D004044 D001186
AND       T0510	// R_P&P Y READY
AND       M01602	// R_P&P Y HOME COMPLETE
OUT       M04102	// R_P&P Y PUT POS
; L135
LOADD=    D004046 D001186
AND       T0510	// R_P&P Y READY
AND       M01602	// R_P&P Y HOME COMPLETE
OUT       M04103	// R_P&P 2D POS
// ----------------------------------------------------------------------------------
// 
// ----  < 11_R_1st ROTATE R >       SERVO MOTOR STATUS  HOME Search
// 
// ----------------------------------------------------------------------------------
; L137
LOAD      D001200.0	// R_1-1 ROT R CTRL RDY
AND       D001200.2	// R_1-1 ROT R SVD ON
AND NOT   D001200.6	// R_1-1 ROT R SVD BUSY
AND NOT   D001200.A	// R_1-1 ROT R WARNING
AND NOT   D001200.B	// R_1-1 ROT R MODULE ERR
AND NOT   D001200.C	// R_1-1 ROT R SVD ERR
AND NOT   M0161A	// R_1-1 ROT R S4th
AND NOT   M00713	// R_1-1 ROT R NOT MV
AND NOT   M0161F	// R_1-1 ROT R MOVE HOLD
OUT       M01610	// R_1-1 ROT R READY
; L138
LOAD      M01610	// R_1-1 ROT R READY
TON       T0511 2	// R_1-1 ROT R READY
TON       T0711 20	// R_1-1 ROT R READY 2s

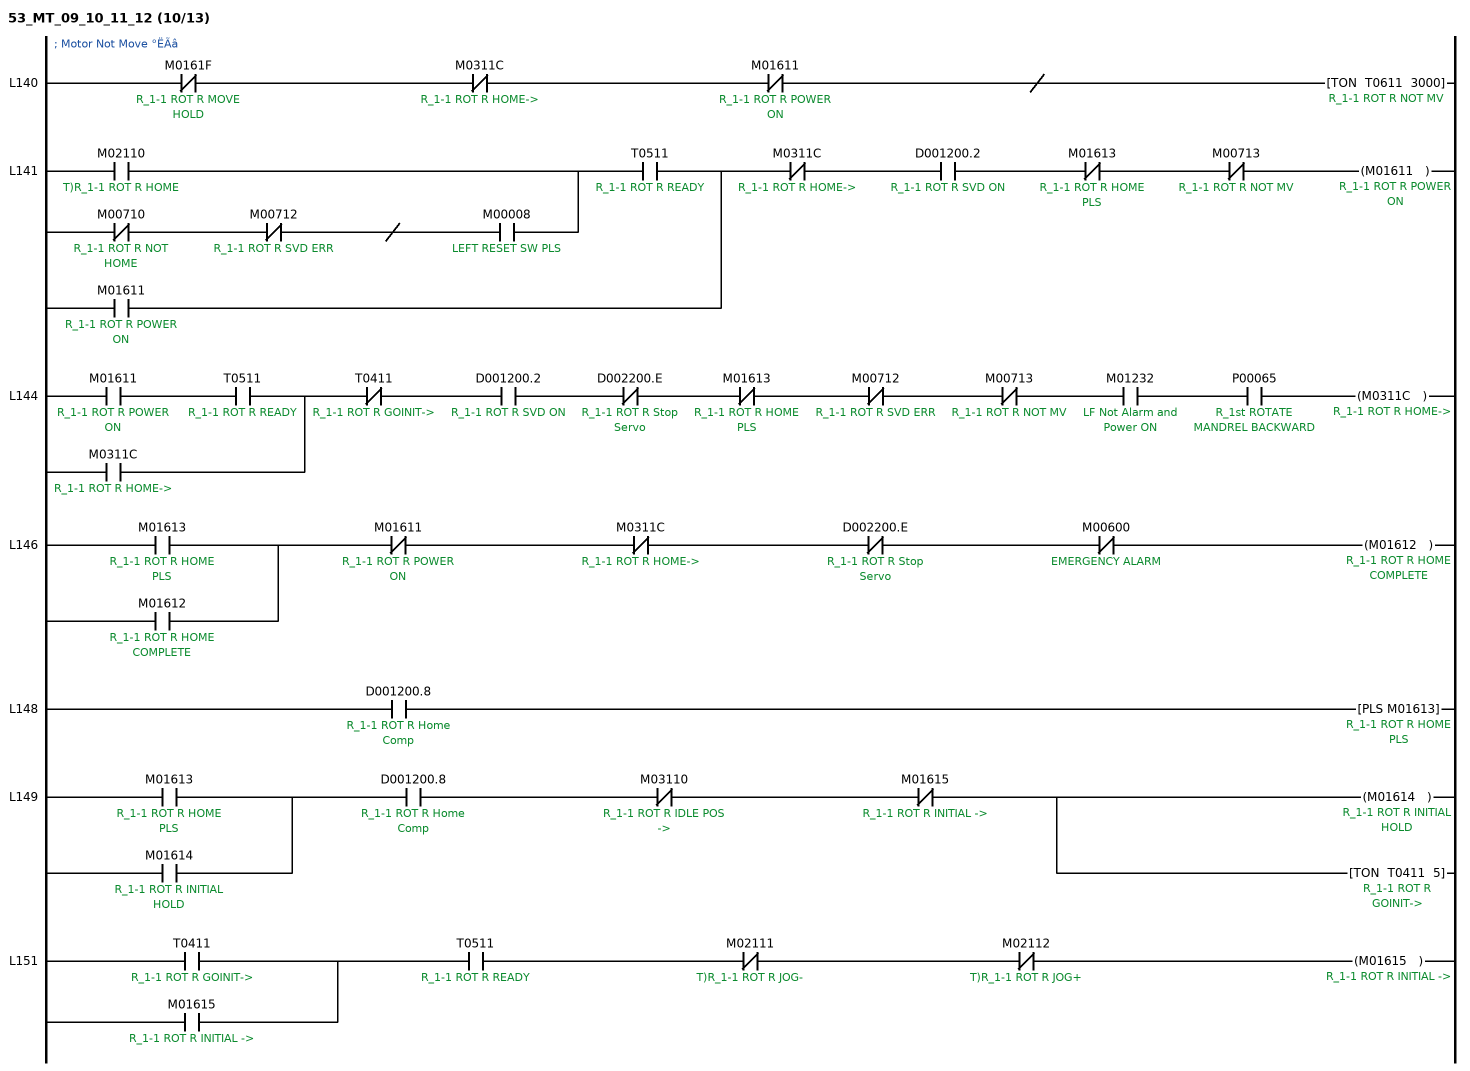
; L140
LOAD NOT  M0161F	// R_1-1 ROT R MOVE HOLD
AND NOT   M0311C	// R_1-1 ROT R HOME->
AND NOT   M01611	// R_1-1 ROT R POWER ON
NOT
TON       T0611 3000	// R_1-1 ROT R NOT MV
// output comment: Motor Not Move °ËÃâ
; L141
LOAD      M02110	// T)R_1-1 ROT R HOME
LOAD NOT  M00710	// R_1-1 ROT R NOT HOME
AND NOT   M00712	// R_1-1 ROT R SVD ERR
NOT
AND       M00008	// LEFT RESET SW PLS
OR LOAD
AND       T0511	// R_1-1 ROT R READY
OR        M01611	// R_1-1 ROT R POWER ON
AND NOT   M0311C	// R_1-1 ROT R HOME->
AND       D001200.2	// R_1-1 ROT R SVD ON
AND NOT   M01613	// R_1-1 ROT R HOME PLS
AND NOT   M00713	// R_1-1 ROT R NOT MV
OUT       M01611	// R_1-1 ROT R POWER ON
; L144
LOAD      M01611	// R_1-1 ROT R POWER ON
AND       T0511	// R_1-1 ROT R READY
OR        M0311C	// R_1-1 ROT R HOME->
AND NOT   T0411	// R_1-1 ROT R GOINIT->
AND       D001200.2	// R_1-1 ROT R SVD ON
AND NOT   D002200.E	// R_1-1 ROT R Stop Servo
AND NOT   M01613	// R_1-1 ROT R HOME PLS
AND NOT   M00712	// R_1-1 ROT R SVD ERR
AND NOT   M00713	// R_1-1 ROT R NOT MV
AND       M01232	// LF Not Alarm and Power ON
AND       P00065	// R_1st ROTATE MANDREL BACKWARD
OUT       M0311C	// R_1-1 ROT R HOME->
; L146
LOAD      M01613	// R_1-1 ROT R HOME PLS
OR        M01612	// R_1-1 ROT R HOME COMPLETE
AND NOT   M01611	// R_1-1 ROT R POWER ON
AND NOT   M0311C	// R_1-1 ROT R HOME->
AND NOT   D002200.E	// R_1-1 ROT R Stop Servo
AND NOT   M00600	// EMERGENCY ALARM
OUT       M01612	// R_1-1 ROT R HOME COMPLETE
; L148
LOAD      D001200.8	// R_1-1 ROT R Home Comp
OUTP      M01613	// R_1-1 ROT R HOME PLS
; L149
LOAD      M01613	// R_1-1 ROT R HOME PLS
OR        M01614	// R_1-1 ROT R INITIAL HOLD
AND       D001200.8	// R_1-1 ROT R Home Comp
AND NOT   M03110	// R_1-1 ROT R IDLE POS ->
AND NOT   M01615	// R_1-1 ROT R INITIAL ->
OUT       M01614	// R_1-1 ROT R INITIAL HOLD
TON       T0411 5	// R_1-1 ROT R GOINIT->
; L151
LOAD      T0411	// R_1-1 ROT R GOINIT->
OR        M01615	// R_1-1 ROT R INITIAL ->
AND       T0511	// R_1-1 ROT R READY
AND NOT   M02111	// T)R_1-1 ROT R JOG-
AND NOT   M02112	// T)R_1-1 ROT R JOG+
OUT       M01615	// R_1-1 ROT R INITIAL ->

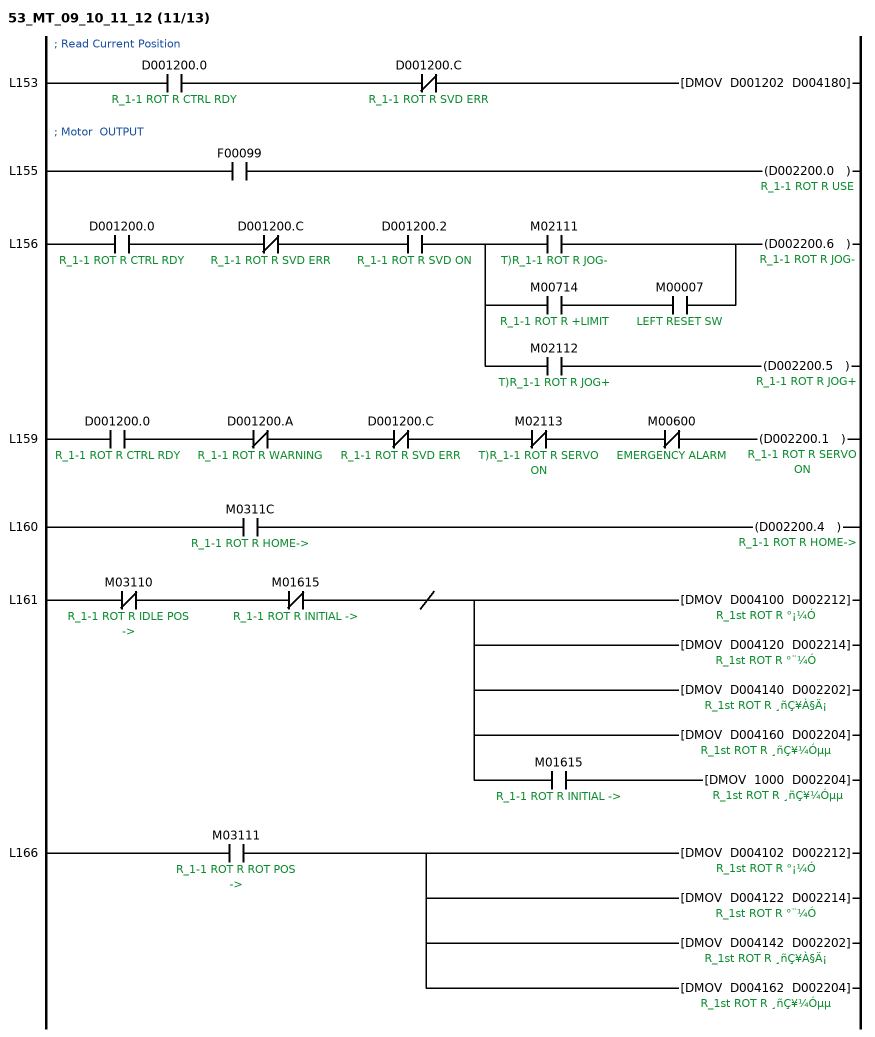
; L153
LOAD      D001200.0	// R_1-1 ROT R CTRL RDY
AND NOT   D001200.C	// R_1-1 ROT R SVD ERR
DMOV      D001202 D004180
// output comment: Read Current Position
//  Motor  OUTPUT
; L155
LOAD      F00099
OUT       D002200.0	// R_1-1 ROT R USE
; L156
LOAD      D001200.0	// R_1-1 ROT R CTRL RDY
AND NOT   D001200.C	// R_1-1 ROT R SVD ERR
AND       D001200.2	// R_1-1 ROT R SVD ON
MPUSH
LOAD      M02111	// T)R_1-1 ROT R JOG-
LOAD      M00714	// R_1-1 ROT R +LIMIT
AND       M00007	// LEFT RESET SW
OR LOAD
AND LOAD
OUT       D002200.6	// R_1-1 ROT R JOG-
MPOP
AND       M02112	// T)R_1-1 ROT R JOG+
OUT       D002200.5	// R_1-1 ROT R JOG+
; L159
LOAD      D001200.0	// R_1-1 ROT R CTRL RDY
AND NOT   D001200.A	// R_1-1 ROT R WARNING
AND NOT   D001200.C	// R_1-1 ROT R SVD ERR
AND NOT   M02113	// T)R_1-1 ROT R SERVO ON
AND NOT   M00600	// EMERGENCY ALARM
OUT       D002200.1	// R_1-1 ROT R SERVO ON
; L160
LOAD      M0311C	// R_1-1 ROT R HOME->
OUT       D002200.4	// R_1-1 ROT R HOME->
; L161
LOAD NOT  M03110	// R_1-1 ROT R IDLE POS ->
AND NOT   M01615	// R_1-1 ROT R INITIAL ->
NOT
DMOV      D004100 D002212	// R_1st ROT R °¡¼Ó
DMOV      D004120 D002214	// R_1st ROT R °¨¼Ó
DMOV      D004140 D002202	// R_1st ROT R ¸ñÇ¥À§Ä¡
DMOV      D004160 D002204	// R_1st ROT R ¸ñÇ¥¼Óµµ
AND       M01615	// R_1-1 ROT R INITIAL ->
DMOV      1000 D002204	// R_1st ROT R ¸ñÇ¥¼Óµµ
; L166
LOAD      M03111	// R_1-1 ROT R ROT POS ->
DMOV      D004102 D002212	// R_1st ROT R °¡¼Ó
DMOV      D004122 D002214	// R_1st ROT R °¨¼Ó
DMOV      D004142 D002202	// R_1st ROT R ¸ñÇ¥À§Ä¡
DMOV      D004162 D002204	// R_1st ROT R ¸ñÇ¥¼Óµµ

